ABB RobotStudio station: CellaRobot1.rspag

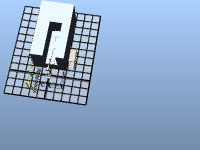
--- station ---
Station CellaRobot (saved by RobotStudio 7.0.8504.151)
Controller IRB_4600_40kg_2.55m
  mechanical unit ROB_1: IRB4600_40_255_C_01, 6 joints, base frame (0, 0, 0) mm
Layout (positions relative to the parent item):
  - IRB4600_40_255_C_01 [mechanism, from Robots\IRB4600_40_255_C_G_01.rslib] at (0, 0, 0) mm; joint values [0, 0, 0, 0, 0.5236, 0] (rad or m)
  - NHX8000 [mechanism, from ADD_Library\NHX8000.rslib] at (0, 0, 0) mm; joint values [2.6, 2] (rad or m)
  - FenceCreator [smart component, from ADD_Library\Recinzione Parametrizzabile.rslib] at (-1991.18, 2102.12, 0) mm
      properties: LengthXside1=3000; LengthYside1=-600; LengthXside2=0; LengthYside2=0; LengthYside3=0; FenceColor=Yellow
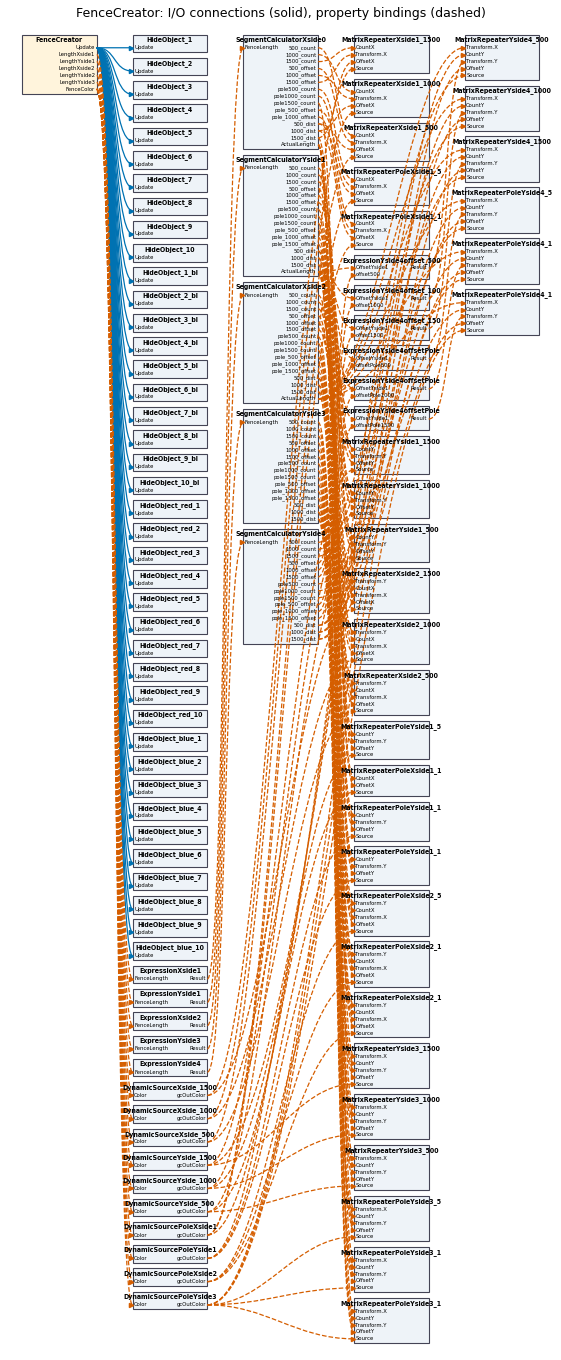
      connections:
        FenceCreator.Update -> HideObject_1.Update
        FenceCreator.Update -> HideObject_2.Update
        FenceCreator.Update -> HideObject_3.Update
        FenceCreator.Update -> HideObject_4.Update
        FenceCreator.Update -> HideObject_5.Update
        FenceCreator.Update -> HideObject_6.Update
        FenceCreator.Update -> HideObject_7.Update
        FenceCreator.Update -> HideObject_8.Update
        FenceCreator.Update -> HideObject_9.Update
        FenceCreator.Update -> HideObject_10.Update
        FenceCreator.Update -> HideObject_1_bl.Update
        FenceCreator.Update -> HideObject_2_bl.Update
        FenceCreator.Update -> HideObject_3_bl.Update
        FenceCreator.Update -> HideObject_4_bl.Update
        FenceCreator.Update -> HideObject_5_bl.Update
        FenceCreator.Update -> HideObject_6_bl.Update
        FenceCreator.Update -> HideObject_7_bl.Update
        FenceCreator.Update -> HideObject_8_bl.Update
        FenceCreator.Update -> HideObject_9_bl.Update
        FenceCreator.Update -> HideObject_10_bl.Update
        FenceCreator.Update -> HideObject_red_1.Update
        FenceCreator.Update -> HideObject_red_2.Update
        FenceCreator.Update -> HideObject_red_3.Update
        FenceCreator.Update -> HideObject_red_4.Update
        FenceCreator.Update -> HideObject_red_5.Update
        FenceCreator.Update -> HideObject_red_6.Update
        FenceCreator.Update -> HideObject_red_7.Update
        FenceCreator.Update -> HideObject_red_8.Update
        FenceCreator.Update -> HideObject_red_9.Update
        FenceCreator.Update -> HideObject_red_10.Update
        FenceCreator.Update -> HideObject_blue_1.Update
        FenceCreator.Update -> HideObject_blue_2.Update
        FenceCreator.Update -> HideObject_blue_3.Update
        FenceCreator.Update -> HideObject_blue_4.Update
        FenceCreator.Update -> HideObject_blue_5.Update
        FenceCreator.Update -> HideObject_blue_6.Update
        FenceCreator.Update -> HideObject_blue_7.Update
        FenceCreator.Update -> HideObject_blue_8.Update
        FenceCreator.Update -> HideObject_blue_9.Update
        FenceCreator.Update -> HideObject_blue_10.Update
        FenceCreator.LengthXside1 => ExpressionXside1.FenceLength
        ExpressionXside1.Result => SegmentCalculatorXside0.FenceLength
        SegmentCalculatorXside0.500_count => MatrixRepeaterXside1_500.CountX
        SegmentCalculatorXside0.1000_count => MatrixRepeaterXside1_1000.CountX
        SegmentCalculatorXside0.1500_count => MatrixRepeaterXside1_1500.CountX
        SegmentCalculatorXside0.500_offset => MatrixRepeaterXside1_500.Transform.X
        SegmentCalculatorXside0.1000_offset => MatrixRepeaterXside1_1000.Transform.X
        SegmentCalculatorXside0.1500_offset => MatrixRepeaterXside1_1500.Transform.X
        SegmentCalculatorXside0.pole500_count => MatrixRepeaterPoleXside1_500.CountX
        SegmentCalculatorXside0.pole1000_count => MatrixRepeaterPoleXside1_1000.CountX
        SegmentCalculatorXside0.pole1500_count => MatrixRepeaterPoleXside1_1500.CountX
        SegmentCalculatorXside0.pole_500_offset => MatrixRepeaterPoleXside1_500.Transform.X
        SegmentCalculatorXside0.pole_1000_offset => MatrixRepeaterPoleXside1_1000.Transform.X
        SegmentCalculatorXside0.500_dist => MatrixRepeaterXside1_500.OffsetX
        SegmentCalculatorXside0.500_dist => MatrixRepeaterPoleXside1_500.OffsetX
        SegmentCalculatorXside0.1000_dist => MatrixRepeaterXside1_1000.OffsetX
        SegmentCalculatorXside0.1000_dist => MatrixRepeaterPoleXside1_1000.OffsetX
        SegmentCalculatorXside0.1500_dist => MatrixRepeaterXside1_1500.OffsetX
        SegmentCalculatorXside0.1500_dist => MatrixRepeaterPoleXside1_1500.OffsetX
        SegmentCalculatorXside0.ActualLength => MatrixRepeaterYside3_500.Transform.X
        SegmentCalculatorXside0.ActualLength => MatrixRepeaterYside3_1000.Transform.X
        SegmentCalculatorXside0.ActualLength => MatrixRepeaterYside3_1500.Transform.X
        SegmentCalculatorXside0.ActualLength => MatrixRepeaterPoleYside3_500.Transform.X
        SegmentCalculatorXside0.ActualLength => MatrixRepeaterPoleYside3_1000.Transform.X
        SegmentCalculatorXside0.ActualLength => MatrixRepeaterPoleYside3_1500.Transform.X
        FenceCreator.LengthYside1 => ExpressionYside1.FenceLength
        ExpressionYside1.Result => SegmentCalculatorYside1.FenceLength
        SegmentCalculatorYside1.500_count => MatrixRepeaterYside1_500.CountY
        SegmentCalculatorYside1.1000_count => MatrixRepeaterYside1_1000.CountY
        SegmentCalculatorYside1.1500_count => MatrixRepeaterYside1_1500.CountY
        SegmentCalculatorYside1.500_offset => MatrixRepeaterYside1_500.Transform.Y
        SegmentCalculatorYside1.1000_offset => MatrixRepeaterYside1_1000.Transform.Y
        SegmentCalculatorYside1.1500_offset => MatrixRepeaterYside1_1500.Transform.Y
        SegmentCalculatorYside1.pole500_count => MatrixRepeaterPoleYside1_500.CountY
        SegmentCalculatorYside1.pole1000_count => MatrixRepeaterPoleYside1_1000.CountY
        SegmentCalculatorYside1.pole1500_count => MatrixRepeaterPoleYside1_1500.CountY
        SegmentCalculatorYside1.pole_500_offset => MatrixRepeaterPoleYside1_500.Transform.Y
        SegmentCalculatorYside1.pole_1000_offset => MatrixRepeaterPoleYside1_1000.Transform.Y
        SegmentCalculatorYside1.pole_1500_offset => MatrixRepeaterPoleYside1_1500.Transform.Y
        SegmentCalculatorYside1.500_dist => MatrixRepeaterYside1_500.OffsetY
        SegmentCalculatorYside1.500_dist => MatrixRepeaterPoleYside1_500.OffsetY
        SegmentCalculatorYside1.1000_dist => MatrixRepeaterYside1_1000.OffsetY
        SegmentCalculatorYside1.1000_dist => MatrixRepeaterPoleYside1_1000.OffsetY
        SegmentCalculatorYside1.1500_dist => MatrixRepeaterYside1_1500.OffsetY
        SegmentCalculatorYside1.1500_dist => MatrixRepeaterPoleYside1_1500.OffsetY
        SegmentCalculatorYside1.ActualLength => MatrixRepeaterXside2_500.Transform.Y
        SegmentCalculatorYside1.ActualLength => MatrixRepeaterXside2_1000.Transform.Y
        SegmentCalculatorYside1.ActualLength => MatrixRepeaterXside2_1500.Transform.Y
        SegmentCalculatorYside1.ActualLength => MatrixRepeaterPoleXside2_500.Transform.Y
        SegmentCalculatorYside1.ActualLength => MatrixRepeaterPoleXside2_1000.Transform.Y
        SegmentCalculatorYside1.ActualLength => MatrixRepeaterPoleXside2_1500.Transform.Y
        SegmentCalculatorYside1.ActualLength => ExpressionYside4offset_500.OffsetYside1
        SegmentCalculatorYside1.ActualLength => ExpressionYside4offset_1000.OffsetYside1
        SegmentCalculatorYside1.ActualLength => ExpressionYside4offset_1500.OffsetYside1
        SegmentCalculatorYside1.ActualLength => ExpressionYside4offsetPole_500.OffsetYside1
        SegmentCalculatorYside1.ActualLength => ExpressionYside4offsetPole_1000.OffsetYside1
        SegmentCalculatorYside1.ActualLength => ExpressionYside4offsetPole_1500.OffsetYside1
        FenceCreator.LengthXside2 => ExpressionXside2.FenceLength
        ExpressionXside2.Result => SegmentCalculatorXside2.FenceLength
        SegmentCalculatorXside2.500_count => MatrixRepeaterXside2_500.CountX
        SegmentCalculatorXside2.1000_count => MatrixRepeaterXside2_1000.CountX
        SegmentCalculatorXside2.1500_count => MatrixRepeaterXside2_1500.CountX
        SegmentCalculatorXside2.500_offset => MatrixRepeaterXside2_500.Transform.X
        SegmentCalculatorXside2.1000_offset => MatrixRepeaterXside2_1000.Transform.X
        SegmentCalculatorXside2.1500_offset => MatrixRepeaterXside2_1500.Transform.X
        SegmentCalculatorXside2.pole500_count => MatrixRepeaterPoleXside2_500.CountX
        SegmentCalculatorXside2.pole1000_count => MatrixRepeaterPoleXside2_1000.CountX
        SegmentCalculatorXside2.pole1500_count => MatrixRepeaterPoleXside2_1500.CountX
        SegmentCalculatorXside2.pole_500_offset => MatrixRepeaterPoleXside2_500.Transform.X
        SegmentCalculatorXside2.pole_1000_offset => MatrixRepeaterPoleXside2_1000.Transform.X
        SegmentCalculatorXside2.pole_1500_offset => MatrixRepeaterPoleXside2_1500.Transform.X
        SegmentCalculatorXside2.500_dist => MatrixRepeaterXside2_500.OffsetX
        SegmentCalculatorXside2.500_dist => MatrixRepeaterPoleXside2_500.OffsetX
        SegmentCalculatorXside2.1000_dist => MatrixRepeaterXside2_1000.OffsetX
        SegmentCalculatorXside2.1000_dist => MatrixRepeaterPoleXside2_1000.OffsetX
        SegmentCalculatorXside2.1500_dist => MatrixRepeaterXside2_1500.OffsetX
        SegmentCalculatorXside2.1500_dist => MatrixRepeaterPoleXside2_1500.OffsetX
        SegmentCalculatorXside2.ActualLength => MatrixRepeaterYside4_500.Transform.X
        SegmentCalculatorXside2.ActualLength => MatrixRepeaterYside4_1000.Transform.X
        SegmentCalculatorXside2.ActualLength => MatrixRepeaterYside4_1500.Transform.X
        SegmentCalculatorXside2.ActualLength => MatrixRepeaterPoleYside4_500.Transform.X
        SegmentCalculatorXside2.ActualLength => MatrixRepeaterPoleYside4_1000.Transform.X
        SegmentCalculatorXside2.ActualLength => MatrixRepeaterPoleYside4_1500.Transform.X
        FenceCreator.LengthYside2 => ExpressionYside3.FenceLength
        ExpressionYside3.Result => SegmentCalculatorYside3.FenceLength
        SegmentCalculatorYside3.500_count => MatrixRepeaterYside3_500.CountY
        SegmentCalculatorYside3.1000_count => MatrixRepeaterYside3_1000.CountY
        SegmentCalculatorYside3.1500_count => MatrixRepeaterYside3_1500.CountY
        SegmentCalculatorYside3.500_offset => MatrixRepeaterYside3_500.Transform.Y
        SegmentCalculatorYside3.1000_offset => MatrixRepeaterYside3_1000.Transform.Y
        SegmentCalculatorYside3.1500_offset => MatrixRepeaterYside3_1500.Transform.Y
        SegmentCalculatorYside3.pole500_count => MatrixRepeaterPoleYside3_500.CountY
        SegmentCalculatorYside3.pole1000_count => MatrixRepeaterPoleYside3_1000.CountY
        SegmentCalculatorYside3.pole1500_count => MatrixRepeaterPoleYside3_1500.CountY
        SegmentCalculatorYside3.pole_500_offset => MatrixRepeaterPoleYside3_500.Transform.Y
        SegmentCalculatorYside3.pole_1000_offset => MatrixRepeaterPoleYside3_1000.Transform.Y
        SegmentCalculatorYside3.pole_1500_offset => MatrixRepeaterPoleYside3_1500.Transform.Y
        SegmentCalculatorYside3.500_dist => MatrixRepeaterYside3_500.OffsetY
        SegmentCalculatorYside3.500_dist => MatrixRepeaterPoleYside3_500.OffsetY
        SegmentCalculatorYside3.1000_dist => MatrixRepeaterYside3_1000.OffsetY
        SegmentCalculatorYside3.1000_dist => MatrixRepeaterPoleYside3_1000.OffsetY
        SegmentCalculatorYside3.1500_dist => MatrixRepeaterYside3_1500.OffsetY
        SegmentCalculatorYside3.1500_dist => MatrixRepeaterPoleYside3_1500.OffsetY
        FenceCreator.LengthYside3 => ExpressionYside4.FenceLength
        ExpressionYside4.Result => SegmentCalculatorYside4.FenceLength
        SegmentCalculatorYside4.500_count => MatrixRepeaterYside4_500.CountY
        SegmentCalculatorYside4.1000_count => MatrixRepeaterYside4_1000.CountY
        SegmentCalculatorYside4.1500_count => MatrixRepeaterYside4_1500.CountY
        SegmentCalculatorYside4.500_offset => ExpressionYside4offset_500.offset500
        SegmentCalculatorYside4.1000_offset => ExpressionYside4offset_1000.offset1000
        SegmentCalculatorYside4.1500_offset => ExpressionYside4offset_1500.offset1500
        SegmentCalculatorYside4.pole500_count => MatrixRepeaterPoleYside4_500.CountY
        SegmentCalculatorYside4.pole1000_count => MatrixRepeaterPoleYside4_1000.CountY
        SegmentCalculatorYside4.pole1500_count => MatrixRepeaterPoleYside4_1500.CountY
        SegmentCalculatorYside4.pole_500_offset => ExpressionYside4offsetPole_500.offsetPole500
        SegmentCalculatorYside4.pole_1000_offset => ExpressionYside4offsetPole_1000.offsetPole1000
        SegmentCalculatorYside4.pole_1500_offset => ExpressionYside4offsetPole_1500.offsetPole1500
        ExpressionYside4offset_500.Result => MatrixRepeaterYside4_500.Transform.Y
        ExpressionYside4offset_1000.Result => MatrixRepeaterYside4_1000.Transform.Y
        ExpressionYside4offset_1500.Result => MatrixRepeaterYside4_1500.Transform.Y
        ExpressionYside4offsetPole_500.Result => MatrixRepeaterPoleYside4_500.Transform.Y
        ExpressionYside4offsetPole_1000.Result => MatrixRepeaterPoleYside4_1000.Transform.Y
        ExpressionYside4offsetPole_1500.Result => MatrixRepeaterPoleYside4_1500.Transform.Y
        SegmentCalculatorYside4.500_dist => MatrixRepeaterYside4_500.OffsetY
        SegmentCalculatorYside4.500_dist => MatrixRepeaterPoleYside4_500.OffsetY
        SegmentCalculatorYside4.1000_dist => MatrixRepeaterYside4_1000.OffsetY
        SegmentCalculatorYside4.1000_dist => MatrixRepeaterPoleYside4_1000.OffsetY
        SegmentCalculatorYside4.1500_dist => MatrixRepeaterYside4_1500.OffsetY
        SegmentCalculatorYside4.1500_dist => MatrixRepeaterPoleYside4_1500.OffsetY
        FenceCreator.FenceColor => DynamicSourceXside_1500.Color
        DynamicSourceXside_1500.gcOutColor => MatrixRepeaterXside1_1500.Source
        DynamicSourceXside_1500.gcOutColor => MatrixRepeaterXside2_1500.Source
        FenceCreator.FenceColor => DynamicSourceXside_1000.Color
        DynamicSourceXside_1000.gcOutColor => MatrixRepeaterXside1_1000.Source
        DynamicSourceXside_1000.gcOutColor => MatrixRepeaterXside2_1000.Source
        FenceCreator.FenceColor => DynamicSourceXside_500.Color
        DynamicSourceXside_500.gcOutColor => MatrixRepeaterXside1_500.Source
        DynamicSourceXside_500.gcOutColor => MatrixRepeaterXside2_500.Source
        FenceCreator.FenceColor => DynamicSourceYside_1500.Color
        DynamicSourceYside_1500.gcOutColor => MatrixRepeaterYside1_1500.Source
        DynamicSourceYside_1500.gcOutColor => MatrixRepeaterYside3_1500.Source
        DynamicSourceYside_1500.gcOutColor => MatrixRepeaterYside4_1500.Source
        FenceCreator.FenceColor => DynamicSourceYside_1000.Color
        DynamicSourceYside_1000.gcOutColor => MatrixRepeaterYside1_1000.Source
        DynamicSourceYside_1000.gcOutColor => MatrixRepeaterYside3_1000.Source
        DynamicSourceYside_1000.gcOutColor => MatrixRepeaterYside4_1000.Source
        FenceCreator.FenceColor => DynamicSourceYside_500.Color
        DynamicSourceYside_500.gcOutColor => MatrixRepeaterYside1_500.Source
        DynamicSourceYside_500.gcOutColor => MatrixRepeaterYside3_500.Source
        DynamicSourceYside_500.gcOutColor => MatrixRepeaterYside4_500.Source
        FenceCreator.FenceColor => DynamicSourcePoleXside1.Color
        DynamicSourcePoleXside1.gcOutColor => MatrixRepeaterPoleXside1_1500.Source
        DynamicSourcePoleXside1.gcOutColor => MatrixRepeaterPoleXside1_1000.Source
        DynamicSourcePoleXside1.gcOutColor => MatrixRepeaterPoleXside1_500.Source
        FenceCreator.FenceColor => DynamicSourcePoleYside1.Color
        DynamicSourcePoleYside1.gcOutColor => MatrixRepeaterPoleYside1_1500.Source
        DynamicSourcePoleYside1.gcOutColor => MatrixRepeaterPoleYside1_1000.Source
        DynamicSourcePoleYside1.gcOutColor => MatrixRepeaterPoleYside1_500.Source
        FenceCreator.FenceColor => DynamicSourcePoleXside2.Color
        DynamicSourcePoleXside2.gcOutColor => MatrixRepeaterPoleXside2_1500.Source
        DynamicSourcePoleXside2.gcOutColor => MatrixRepeaterPoleXside2_1000.Source
        DynamicSourcePoleXside2.gcOutColor => MatrixRepeaterPoleXside2_500.Source
        FenceCreator.FenceColor => DynamicSourcePoleYside3.Color
        DynamicSourcePoleYside3.gcOutColor => MatrixRepeaterPoleYside3_1500.Source
        DynamicSourcePoleYside3.gcOutColor => MatrixRepeaterPoleYside3_1000.Source
        DynamicSourcePoleYside3.gcOutColor => MatrixRepeaterPoleYside3_500.Source
        DynamicSourcePoleYside3.gcOutColor => MatrixRepeaterPoleYside4_1500.Source
        DynamicSourcePoleYside3.gcOutColor => MatrixRepeaterPoleYside4_1000.Source
        DynamicSourcePoleYside3.gcOutColor => MatrixRepeaterPoleYside4_500.Source
    - ExpressionXside1 [smart component, from ADD_Library\Recinzione Parametrizzabile.rslib]
        properties: Expression=FenceLength/1000; Result=3; FenceLength=3000
    - MatrixRepeaterXside1_1500 [smart component, from ADD_Library\Recinzione Parametrizzabile.rslib]
        properties: Source=Panel 2000x1500 X ye; CountX=2; CountY=1; CountZ=1; OffsetX=1.5; OffsetY=0; OffsetZ=0
      - Panel 2000x1500 X ye [part, from ADD_Library\Recinzione Parametrizzabile.rslib]
      - Panel 2000x1500 X ye [part, from ADD_Library\Recinzione Parametrizzabile.rslib] at (1500, 0, 0) mm
    - Panel 2000x1000 X ye [part, from ADD_Library\Recinzione Parametrizzabile.rslib]
    - Panel 2000x500 X ye [part, from ADD_Library\Recinzione Parametrizzabile.rslib]
    - Panel 2000x1500 X ye [part, from ADD_Library\Recinzione Parametrizzabile.rslib]
    - MatrixRepeaterXside1_1000 [smart component, from ADD_Library\Recinzione Parametrizzabile.rslib] at (3000, 0, 0) mm
        properties: Source=Panel 2000x1000 X ye; CountX=0; CountY=1; CountZ=1; OffsetX=1; OffsetY=0; OffsetZ=0
    - MatrixRepeaterXside1_500 [smart component, from ADD_Library\Recinzione Parametrizzabile.rslib] at (3000, 0, 0) mm
        properties: Source=Panel 2000x500 X ye; CountX=0; CountY=1; CountZ=1; OffsetX=0.5; OffsetY=0; OffsetZ=0
    - MatrixRepeaterPoleXside1_1000 [smart component, from ADD_Library\Recinzione Parametrizzabile.rslib] at (4000, 0, 0) mm
        properties: Source=Pole ye; CountX=0; CountY=1; CountZ=1; OffsetX=1; OffsetY=0; OffsetZ=0
    - Pole ye [part, from ADD_Library\Recinzione Parametrizzabile.rslib]
    - SegmentCalculatorXside0 [smart component, from ADD_Library\Recinzione Parametrizzabile.rslib]
        properties: FenceLength=3; ActualLength=3; 1500_dist=1.5; 1000_dist=1; 500_dist=0.5; 1500_offset=0; 1000_offset=3; 500_offset=3; pole_1500_offset=0; pole_1000_offset=4; pole_500_offset=3.5; 1500_count=2; 1000_count=0; 500_count=0; pole1500_count=3; pole1000_count=0; pole500_count=0; SideNo=0
    - MatrixRepeaterPoleXside1_1500 [smart component, from ADD_Library\Recinzione Parametrizzabile.rslib]
        properties: Source=Pole ye; CountX=3; CountY=1; CountZ=1; OffsetX=1.5; OffsetY=0; OffsetZ=1
      - Pole ye [part, from ADD_Library\Recinzione Parametrizzabile.rslib]
      - Pole ye [part, from ADD_Library\Recinzione Parametrizzabile.rslib] at (1500, 0, 0) mm
      - Pole ye [part, from ADD_Library\Recinzione Parametrizzabile.rslib] at (3000, 0, 0) mm
    - MatrixRepeaterPoleXside1_500 [smart component, from ADD_Library\Recinzione Parametrizzabile.rslib] at (3500, 0, 0) mm
        properties: Source=Pole ye; CountX=0; CountY=1; CountZ=1; OffsetX=0.5; OffsetY=0; OffsetZ=0
    - Panel 2000x1000 Y ye [part, from ADD_Library\Recinzione Parametrizzabile.rslib]
    - Panel 2000x500 Y ye [part, from ADD_Library\Recinzione Parametrizzabile.rslib]
    - Panel 2000x1500 Y ye [part, from ADD_Library\Recinzione Parametrizzabile.rslib]
    - ExpressionYside1 [smart component, from ADD_Library\Recinzione Parametrizzabile.rslib]
        properties: Expression=FenceLength/1000; Result=-0.6; FenceLength=-600
    - MatrixRepeaterYside1_1500 [smart component, from ADD_Library\Recinzione Parametrizzabile.rslib] at (0, -1500, 0) mm
        properties: Source=Panel 2000x1500 Y ye; CountX=1; CountY=0; CountZ=1; OffsetX=0; OffsetY=-1.5; OffsetZ=0
    - MatrixRepeaterYside1_1000 [smart component, from ADD_Library\Recinzione Parametrizzabile.rslib] at (0, -1000, 0) mm
        properties: Source=Panel 2000x1000 Y ye; CountX=1; CountY=0; CountZ=1; OffsetX=0; OffsetY=-1; OffsetZ=0
    - MatrixRepeaterYside1_500 [smart component, from ADD_Library\Recinzione Parametrizzabile.rslib] at (0, -500, 0) mm
        properties: Source=Panel 2000x500 Y ye; CountX=1; CountY=1; CountZ=1; OffsetX=0; OffsetY=-0.5; OffsetZ=0
      - Panel 2000x500 Y ye [part, from ADD_Library\Recinzione Parametrizzabile.rslib]
    - PoleYside1 ye [part, from ADD_Library\Recinzione Parametrizzabile.rslib]
    - MatrixRepeaterPoleYside1_1500 [smart component, from ADD_Library\Recinzione Parametrizzabile.rslib] at (0, 1500, 0) mm
        properties: Source=PoleYside1 ye; CountX=1; CountY=0; CountZ=1; OffsetX=0; OffsetY=-1.5; OffsetZ=0
    - SegmentCalculatorYside1 [smart component, from ADD_Library\Recinzione Parametrizzabile.rslib]
        properties: FenceLength=-0.6; ActualLength=-0.5; 1500_dist=-1.5; 1000_dist=-1; 500_dist=-0.5; 1500_offset=-1.5; 1000_offset=-1; 500_offset=-0.5; pole_1500_offset=1.5; pole_1000_offset=1; pole_500_offset=-0.5; 1500_count=0; 1000_count=0; 500_count=1; pole1500_count=0; pole1000_count=0; pole500_count=1; SideNo=1
    - MatrixRepeaterPoleYside1_1000 [smart component, from ADD_Library\Recinzione Parametrizzabile.rslib] at (0, 1000, 0) mm
        properties: Source=PoleYside1 ye; CountX=1; CountY=0; CountZ=1; OffsetX=0; OffsetY=-1; OffsetZ=0
    - MatrixRepeaterPoleYside1_500 [smart component, from ADD_Library\Recinzione Parametrizzabile.rslib] at (0, -500, 0) mm
        properties: Source=PoleYside1 ye; CountX=1; CountY=1; CountZ=1; OffsetX=0; OffsetY=-0.5; OffsetZ=0
      - PoleYside1 ye [part, from ADD_Library\Recinzione Parametrizzabile.rslib]
    - PoleXside2 ye [part, from ADD_Library\Recinzione Parametrizzabile.rslib]
    - PoleYside3 ye [part, from ADD_Library\Recinzione Parametrizzabile.rslib]
    - ExpressionXside2 [smart component, from ADD_Library\Recinzione Parametrizzabile.rslib]
        properties: Expression=FenceLength/1000; Result=0; FenceLength=0
    - SegmentCalculatorXside2 [smart component, from ADD_Library\Recinzione Parametrizzabile.rslib]
        properties: FenceLength=0; ActualLength=0; 1500_dist=1.5; 1000_dist=1; 500_dist=0.5; 1500_offset=0; 1000_offset=0; 500_offset=0; pole_1500_offset=1.5; pole_1000_offset=1; pole_500_offset=0; 1500_count=0; 1000_count=0; 500_count=0; pole1500_count=0; pole1000_count=0; pole500_count=0; SideNo=2
    - MatrixRepeaterXside2_1500 [smart component, from ADD_Library\Recinzione Parametrizzabile.rslib] at (0, -500, 0) mm
        properties: Source=Panel 2000x1500 X ye; CountX=0; CountY=1; CountZ=1; OffsetX=1.5; OffsetY=0; OffsetZ=0
    - MatrixRepeaterXside2_1000 [smart component, from ADD_Library\Recinzione Parametrizzabile.rslib] at (0, -500, 0) mm
        properties: Source=Panel 2000x1000 X ye; CountX=0; CountY=1; CountZ=1; OffsetX=1; OffsetY=0; OffsetZ=0
    - MatrixRepeaterXside2_500 [smart component, from ADD_Library\Recinzione Parametrizzabile.rslib] at (0, -500, 0) mm
        properties: Source=Panel 2000x500 X ye; CountX=0; CountY=1; CountZ=1; OffsetX=0.5; OffsetY=0; OffsetZ=0
    - MatrixRepeaterPoleXside2_1500 [smart component, from ADD_Library\Recinzione Parametrizzabile.rslib] at (1500, -500, 0) mm
        properties: Source=PoleXside2 ye; CountX=0; CountY=1; CountZ=1; OffsetX=1.5; OffsetY=0; OffsetZ=0
    - MatrixRepeaterPoleXside2_1000 [smart component, from ADD_Library\Recinzione Parametrizzabile.rslib] at (1000, -500, 0) mm
        properties: Source=PoleXside2 ye; CountX=0; CountY=1; CountZ=1; OffsetX=1; OffsetY=0; OffsetZ=0
    - MatrixRepeaterPoleXside2_500 [smart component, from ADD_Library\Recinzione Parametrizzabile.rslib] at (0, -500, 0) mm
        properties: Source=PoleXside2 ye; CountX=0; CountY=1; CountZ=1; OffsetX=0.5; OffsetY=0; OffsetZ=0
    - SegmentCalculatorYside3 [smart component, from ADD_Library\Recinzione Parametrizzabile.rslib]
        properties: FenceLength=0; ActualLength=0; 1500_dist=1.5; 1000_dist=1; 500_dist=0.5; 1500_offset=0; 1000_offset=0; 500_offset=0; pole_1500_offset=-1.5; pole_1000_offset=-2.5; pole_500_offset=0; 1500_count=0; 1000_count=0; 500_count=0; pole1500_count=0; pole1000_count=0; pole500_count=0; SideNo=3
    - ExpressionYside3 [smart component, from ADD_Library\Recinzione Parametrizzabile.rslib]
        properties: Expression=FenceLength/1000; Result=0; FenceLength=0
    - MatrixRepeaterYside3_1500 [smart component, from ADD_Library\Recinzione Parametrizzabile.rslib] at (3000, 0, 0) mm
        properties: Source=Panel 2000x1500 Y ye; CountX=1; CountY=0; CountZ=1; OffsetX=0; OffsetY=1.5; OffsetZ=0
    - MatrixRepeaterYside3_1000 [smart component, from ADD_Library\Recinzione Parametrizzabile.rslib] at (3000, 0, 0) mm
        properties: Source=Panel 2000x1000 Y ye; CountX=1; CountY=0; CountZ=1; OffsetX=0; OffsetY=1; OffsetZ=0
    - MatrixRepeaterYside3_500 [smart component, from ADD_Library\Recinzione Parametrizzabile.rslib] at (3000, 0, 0) mm
        properties: Source=Panel 2000x500 Y ye; CountX=1; CountY=0; CountZ=1; OffsetX=0; OffsetY=0.5; OffsetZ=0
    - MatrixRepeaterPoleYside3_1500 [smart component, from ADD_Library\Recinzione Parametrizzabile.rslib] at (3000, -1500, 0) mm
        properties: Source=PoleYside3 ye; CountX=1; CountY=0; CountZ=1; OffsetX=0; OffsetY=1.5; OffsetZ=0
    - MatrixRepeaterPoleYside3_1000 [smart component, from ADD_Library\Recinzione Parametrizzabile.rslib] at (3000, -2500, 0) mm
        properties: Source=PoleYside3 ye; CountX=1; CountY=0; CountZ=1; OffsetX=0; OffsetY=1; OffsetZ=0
    - MatrixRepeaterPoleYside3_500 [smart component, from ADD_Library\Recinzione Parametrizzabile.rslib] at (3000, 0, 0) mm
        properties: Source=PoleYside3 ye; CountX=1; CountY=0; CountZ=1; OffsetX=0; OffsetY=0.5; OffsetZ=0
    - ExpressionYside4 [smart component, from ADD_Library\Recinzione Parametrizzabile.rslib]
        properties: Expression=FenceLength/1000; Result=0; FenceLength=0
    - SegmentCalculatorYside4 [smart component, from ADD_Library\Recinzione Parametrizzabile.rslib]
        properties: FenceLength=0; ActualLength=0; 1500_dist=1.5; 1000_dist=1; 500_dist=0.5; 1500_offset=0; 1000_offset=0; 500_offset=0; pole_1500_offset=1.5; pole_1000_offset=2.5; pole_500_offset=0; 1500_count=0; 1000_count=0; 500_count=0; pole1500_count=0; pole1000_count=0; pole500_count=0; SideNo=4
    - MatrixRepeaterYside4_1500 [smart component, from ADD_Library\Recinzione Parametrizzabile.rslib] at (0, -500, 0) mm
        properties: Source=Panel 2000x1500 Y ye; CountX=1; CountY=0; CountZ=1; OffsetX=0; OffsetY=1.5; OffsetZ=0
    - ExpressionYside4offset_500 [smart component, from ADD_Library\Recinzione Parametrizzabile.rslib]
        properties: Expression=OffsetYside1+offset500; Result=-0.5; OffsetYside1=-0.5; offset500=0
    - ExpressionYside4offset_1000 [smart component, from ADD_Library\Recinzione Parametrizzabile.rslib]
        properties: Expression=OffsetYside1+offset1000; Result=-0.5; OffsetYside1=-0.5; offset1000=0
    - ExpressionYside4offset_1500 [smart component, from ADD_Library\Recinzione Parametrizzabile.rslib]
        properties: Expression=OffsetYside1+offset1500; Result=-0.5; OffsetYside1=-0.5; offset1500=0
    - MatrixRepeaterYside4_1000 [smart component, from ADD_Library\Recinzione Parametrizzabile.rslib] at (0, -500, 0) mm
        properties: Source=Panel 2000x1000 Y ye; CountX=1; CountY=0; CountZ=1; OffsetX=0; OffsetY=1; OffsetZ=0
    - MatrixRepeaterYside4_500 [smart component, from ADD_Library\Recinzione Parametrizzabile.rslib] at (0, -500, 0) mm
        properties: Source=Panel 2000x500 Y ye; CountX=1; CountY=0; CountZ=1; OffsetX=0; OffsetY=0.5; OffsetZ=0
    - ExpressionYside4offsetPole_500 [smart component, from ADD_Library\Recinzione Parametrizzabile.rslib]
        properties: Expression=OffsetYside1+offsetPole500; Result=-0.5; OffsetYside1=-0.5; offsetPole500=0
    - ExpressionYside4offsetPole_1000 [smart component, from ADD_Library\Recinzione Parametrizzabile.rslib]
        properties: Expression=OffsetYside1+offsetPole1000; Result=2; OffsetYside1=-0.5; offsetPole1000=2.5
    - ExpressionYside4offsetPole_1500 [smart component, from ADD_Library\Recinzione Parametrizzabile.rslib]
        properties: Expression=OffsetYside1+offsetPole1500; Result=1; OffsetYside1=-0.5; offsetPole1500=1.5
    - MatrixRepeaterPoleYside4_500 [smart component, from ADD_Library\Recinzione Parametrizzabile.rslib] at (0, -500, 0) mm
        properties: Source=PoleYside3 ye; CountX=1; CountY=0; CountZ=1; OffsetX=0; OffsetY=0.5; OffsetZ=0
    - MatrixRepeaterPoleYside4_1000 [smart component, from ADD_Library\Recinzione Parametrizzabile.rslib] at (0, 2000, 0) mm
        properties: Source=PoleYside3 ye; CountX=1; CountY=0; CountZ=1; OffsetX=0; OffsetY=1; OffsetZ=0
    - MatrixRepeaterPoleYside4_1500 [smart component, from ADD_Library\Recinzione Parametrizzabile.rslib] at (0, 1000, 0) mm
        properties: Source=PoleYside3 ye; CountX=1; CountY=0; CountZ=1; OffsetX=0; OffsetY=1.5; OffsetZ=0
    - HideObject_1 [smart component, from ADD_Library\Recinzione Parametrizzabile.rslib]
        properties: Object=Panel 2000x500 X ye
    - HideObject_2 [smart component, from ADD_Library\Recinzione Parametrizzabile.rslib]
        properties: Object=Panel 2000x1000 X ye
    - HideObject_3 [smart component, from ADD_Library\Recinzione Parametrizzabile.rslib]
        properties: Object=Panel 2000x1500 X ye
    - HideObject_4 [smart component, from ADD_Library\Recinzione Parametrizzabile.rslib]
        properties: Object=Panel 2000x500 Y ye
    - HideObject_5 [smart component, from ADD_Library\Recinzione Parametrizzabile.rslib]
        properties: Object=Panel 2000x1000 Y ye
    - HideObject_6 [smart component, from ADD_Library\Recinzione Parametrizzabile.rslib]
        properties: Object=Panel 2000x1500 Y ye
    - HideObject_7 [smart component, from ADD_Library\Recinzione Parametrizzabile.rslib]
        properties: Object=Pole ye
    - HideObject_8 [smart component, from ADD_Library\Recinzione Parametrizzabile.rslib]
        properties: Object=PoleYside1 ye
    - HideObject_9 [smart component, from ADD_Library\Recinzione Parametrizzabile.rslib]
        properties: Object=PoleXside2 ye
    - HideObject_10 [smart component, from ADD_Library\Recinzione Parametrizzabile.rslib]
        properties: Object=PoleYside3 ye
    - Panel 2000x1000 X bl [part, from ADD_Library\Recinzione Parametrizzabile.rslib]
    - Panel 2000x500 X bl [part, from ADD_Library\Recinzione Parametrizzabile.rslib]
    - Panel 2000x1500 X bl [part, from ADD_Library\Recinzione Parametrizzabile.rslib]
    - Pole bl [part, from ADD_Library\Recinzione Parametrizzabile.rslib]
    - Panel 2000x1000 Y bl [part, from ADD_Library\Recinzione Parametrizzabile.rslib]
    - Panel 2000x500 Y bl [part, from ADD_Library\Recinzione Parametrizzabile.rslib]
    - Panel 2000x1500 Y bl [part, from ADD_Library\Recinzione Parametrizzabile.rslib]
    - PoleYside1 bl [part, from ADD_Library\Recinzione Parametrizzabile.rslib]
    - PoleXside2 bl [part, from ADD_Library\Recinzione Parametrizzabile.rslib]
    - PoleYside3 bl [part, from ADD_Library\Recinzione Parametrizzabile.rslib]
    - DynamicSourceXside_1500 [smart component, from ADD_Library\Recinzione Parametrizzabile.rslib]
        properties: gcBlack=Panel 2000x1500 X bl; gcYellow=Panel 2000x1500 X ye; gcRed=Panel 2000x1500 X red; gcBlue=Panel 2000x1500 X_blue; Color=Yellow; gcOutColor=Panel 2000x1500 X ye
    - DynamicSourceXside_1000 [smart component, from ADD_Library\Recinzione Parametrizzabile.rslib]
        properties: gcBlack=Panel 2000x1000 X bl; gcYellow=Panel 2000x1000 X ye; gcRed=Panel 2000x1000 X red; gcBlue=Panel 2000x1000 X_blue; Color=Yellow; gcOutColor=Panel 2000x1000 X ye
    - DynamicSourceXside_500 [smart component, from ADD_Library\Recinzione Parametrizzabile.rslib]
        properties: gcBlack=Panel 2000x500 X bl; gcYellow=Panel 2000x500 X ye; gcRed=Panel 2000x500 X red; gcBlue=Panel 2000x500 X blue; Color=Yellow; gcOutColor=Panel 2000x500 X ye
    - DynamicSourceYside_1500 [smart component, from ADD_Library\Recinzione Parametrizzabile.rslib]
        properties: gcBlack=Panel 2000x1500 Y bl; gcYellow=Panel 2000x1500 Y ye; gcRed=Panel 2000x1500 Y red; gcBlue=Panel 2000x1500 Y_blue; Color=Yellow; gcOutColor=Panel 2000x1500 Y ye
    - DynamicSourceYside_1000 [smart component, from ADD_Library\Recinzione Parametrizzabile.rslib]
        properties: gcBlack=Panel 2000x1000 Y bl; gcYellow=Panel 2000x1000 Y ye; gcRed=Panel 2000x1000 Y red; gcBlue=Panel 2000x1000 Y_blue; Color=Yellow; gcOutColor=Panel 2000x1000 Y ye
    - DynamicSourceYside_500 [smart component, from ADD_Library\Recinzione Parametrizzabile.rslib]
        properties: gcBlack=Panel 2000x500 Y bl; gcYellow=Panel 2000x500 Y ye; gcRed=Panel 2000x500 Y red; gcBlue=Panel 2000x500 Y blue; Color=Yellow; gcOutColor=Panel 2000x500 Y ye
    - DynamicSourcePoleXside1 [smart component, from ADD_Library\Recinzione Parametrizzabile.rslib]
        properties: gcBlack=Pole bl; gcYellow=Pole ye; gcRed=Pole_red; gcBlue=Pole_blue; Color=Yellow; gcOutColor=Pole ye
    - DynamicSourcePoleYside1 [smart component, from ADD_Library\Recinzione Parametrizzabile.rslib]
        properties: gcBlack=PoleYside1 bl; gcYellow=PoleYside1 ye; gcRed=PoleYside1_red; gcBlue=PoleYside1_blue; Color=Yellow; gcOutColor=PoleYside1 ye
    - DynamicSourcePoleXside2 [smart component, from ADD_Library\Recinzione Parametrizzabile.rslib]
        properties: gcBlack=PoleXside2 bl; gcYellow=PoleXside2 ye; gcRed=PoleXside2_red; gcBlue=PoleXside2_blue; Color=Yellow; gcOutColor=PoleXside2 ye
    - DynamicSourcePoleYside3 [smart component, from ADD_Library\Recinzione Parametrizzabile.rslib]
        properties: gcBlack=PoleYside3 bl; gcYellow=PoleYside3 ye; gcRed=PoleYside3 red; gcBlue=PoleYside3 blue; Color=Yellow; gcOutColor=PoleYside3 ye
    - HideObject_1_bl [smart component, from ADD_Library\Recinzione Parametrizzabile.rslib]
        properties: Object=Panel 2000x1500 X bl
    - HideObject_2_bl [smart component, from ADD_Library\Recinzione Parametrizzabile.rslib]
        properties: Object=Panel 2000x1000 X bl
    - HideObject_3_bl [smart component, from ADD_Library\Recinzione Parametrizzabile.rslib]
        properties: Object=Panel 2000x500 X bl
    - HideObject_4_bl [smart component, from ADD_Library\Recinzione Parametrizzabile.rslib]
        properties: Object=Panel 2000x1500 Y bl
    - HideObject_5_bl [smart component, from ADD_Library\Recinzione Parametrizzabile.rslib]
        properties: Object=Panel 2000x1000 Y bl
    - HideObject_6_bl [smart component, from ADD_Library\Recinzione Parametrizzabile.rslib]
        properties: Object=Panel 2000x500 Y bl
    - HideObject_7_bl [smart component, from ADD_Library\Recinzione Parametrizzabile.rslib]
        properties: Object=Pole bl
    - HideObject_8_bl [smart component, from ADD_Library\Recinzione Parametrizzabile.rslib]
        properties: Object=PoleYside1 bl
    - HideObject_9_bl [smart component, from ADD_Library\Recinzione Parametrizzabile.rslib]
        properties: Object=PoleXside2 bl
    - HideObject_10_bl [smart component, from ADD_Library\Recinzione Parametrizzabile.rslib]
        properties: Object=PoleYside3 bl
    - Panel 2000x500 X blue [part, from ADD_Library\Recinzione Parametrizzabile.rslib]
    - Panel 2000x500 X red [part, from ADD_Library\Recinzione Parametrizzabile.rslib]
    - Panel 2000x500 Y blue [part, from ADD_Library\Recinzione Parametrizzabile.rslib]
    - Panel 2000x500 Y red [part, from ADD_Library\Recinzione Parametrizzabile.rslib]
    - Panel 2000x1000 X red [part, from ADD_Library\Recinzione Parametrizzabile.rslib]
    - Panel 2000x1000 X_blue [part, from ADD_Library\Recinzione Parametrizzabile.rslib]
    - Panel 2000x1000 Y red [part, from ADD_Library\Recinzione Parametrizzabile.rslib]
    - Panel 2000x1000 Y_blue [part, from ADD_Library\Recinzione Parametrizzabile.rslib]
    - Panel 2000x1500 X red [part, from ADD_Library\Recinzione Parametrizzabile.rslib]
    - Panel 2000x1500 X_blue [part, from ADD_Library\Recinzione Parametrizzabile.rslib]
    - Panel 2000x1500 Y red [part, from ADD_Library\Recinzione Parametrizzabile.rslib]
    - Panel 2000x1500 Y_blue [part, from ADD_Library\Recinzione Parametrizzabile.rslib]
    - Pole_blue [part, from ADD_Library\Recinzione Parametrizzabile.rslib]
    - Pole_red [part, from ADD_Library\Recinzione Parametrizzabile.rslib]
    - PoleXside2_blue [part, from ADD_Library\Recinzione Parametrizzabile.rslib]
    - PoleXside2_red [part, from ADD_Library\Recinzione Parametrizzabile.rslib]
    - PoleYside1_blue [part, from ADD_Library\Recinzione Parametrizzabile.rslib]
    - PoleYside1_red [part, from ADD_Library\Recinzione Parametrizzabile.rslib]
    - PoleYside3 blue [part, from ADD_Library\Recinzione Parametrizzabile.rslib]
    - PoleYside3 red [part, from ADD_Library\Recinzione Parametrizzabile.rslib]
    - HideObject_red_1 [smart component, from ADD_Library\Recinzione Parametrizzabile.rslib]
        properties: Object=Panel 2000x1500 X red
    - HideObject_red_2 [smart component, from ADD_Library\Recinzione Parametrizzabile.rslib]
        properties: Object=Panel 2000x1500 Y red
    - HideObject_red_3 [smart component, from ADD_Library\Recinzione Parametrizzabile.rslib]
        properties: Object=Panel 2000x1000 X red
    - HideObject_red_4 [smart component, from ADD_Library\Recinzione Parametrizzabile.rslib]
        properties: Object=Panel 2000x1000 Y red
    - HideObject_red_5 [smart component, from ADD_Library\Recinzione Parametrizzabile.rslib]
        properties: Object=Panel 2000x500 X red
    - HideObject_red_6 [smart component, from ADD_Library\Recinzione Parametrizzabile.rslib]
        properties: Object=Panel 2000x500 Y red
    - HideObject_red_7 [smart component, from ADD_Library\Recinzione Parametrizzabile.rslib]
        properties: Object=Pole_red
    - HideObject_red_8 [smart component, from ADD_Library\Recinzione Parametrizzabile.rslib]
        properties: Object=PoleXside2_red
    - HideObject_red_9 [smart component, from ADD_Library\Recinzione Parametrizzabile.rslib]
        properties: Object=PoleYside1_red
    - HideObject_red_10 [smart component, from ADD_Library\Recinzione Parametrizzabile.rslib]
        properties: Object=PoleYside3 red
    - HideObject_blue_1 [smart component, from ADD_Library\Recinzione Parametrizzabile.rslib]
        properties: Object=Panel 2000x1500 X_blue
    - HideObject_blue_2 [smart component, from ADD_Library\Recinzione Parametrizzabile.rslib]
        properties: Object=Panel 2000x1500 Y_blue
    - HideObject_blue_3 [smart component, from ADD_Library\Recinzione Parametrizzabile.rslib]
        properties: Object=Panel 2000x1000 X_blue
    - HideObject_blue_4 [smart component, from ADD_Library\Recinzione Parametrizzabile.rslib]
        properties: Object=Panel 2000x1000 Y_blue
    - HideObject_blue_5 [smart component, from ADD_Library\Recinzione Parametrizzabile.rslib]
        properties: Object=Panel 2000x500 X blue
    - HideObject_blue_6 [smart component, from ADD_Library\Recinzione Parametrizzabile.rslib]
        properties: Object=Panel 2000x500 Y blue
    - HideObject_blue_7 [smart component, from ADD_Library\Recinzione Parametrizzabile.rslib]
        properties: Object=Pole_blue
    - HideObject_blue_8 [smart component, from ADD_Library\Recinzione Parametrizzabile.rslib]
        properties: Object=PoleXside2_blue
    - HideObject_blue_9 [smart component, from ADD_Library\Recinzione Parametrizzabile.rslib]
        properties: Object=PoleYside1_blue
    - HideObject_blue_10 [smart component, from ADD_Library\Recinzione Parametrizzabile.rslib]
        properties: Object=PoleYside3 blue
  - FenceCreator_2 [smart component, from ADD_Library\Recinzione Parametrizzabile.rslib] at (-1501.5, -1896.94, 0) mm
      properties: LengthXside1=2500; LengthYside1=2500; LengthXside2=0; LengthYside2=0; LengthYside3=0; FenceColor=Black
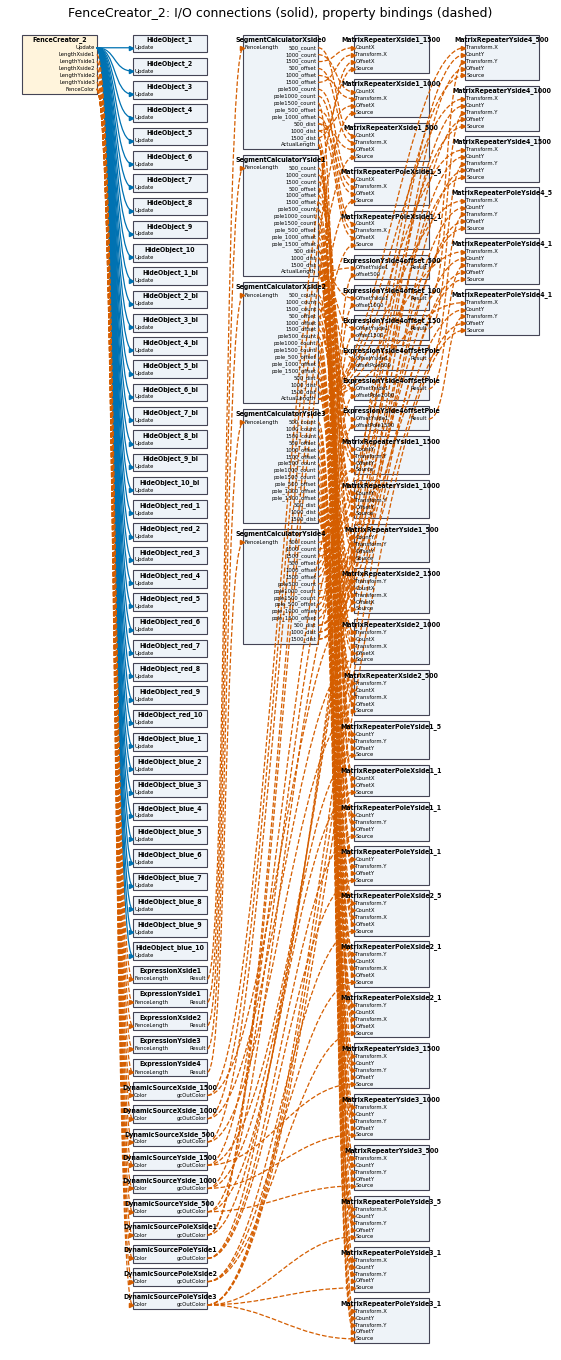
      connections:
        FenceCreator_2.Update -> HideObject_1.Update
        FenceCreator_2.Update -> HideObject_2.Update
        FenceCreator_2.Update -> HideObject_3.Update
        FenceCreator_2.Update -> HideObject_4.Update
        FenceCreator_2.Update -> HideObject_5.Update
        FenceCreator_2.Update -> HideObject_6.Update
        FenceCreator_2.Update -> HideObject_7.Update
        FenceCreator_2.Update -> HideObject_8.Update
        FenceCreator_2.Update -> HideObject_9.Update
        FenceCreator_2.Update -> HideObject_10.Update
        FenceCreator_2.Update -> HideObject_1_bl.Update
        FenceCreator_2.Update -> HideObject_2_bl.Update
        FenceCreator_2.Update -> HideObject_3_bl.Update
        FenceCreator_2.Update -> HideObject_4_bl.Update
        FenceCreator_2.Update -> HideObject_5_bl.Update
        FenceCreator_2.Update -> HideObject_6_bl.Update
        FenceCreator_2.Update -> HideObject_7_bl.Update
        FenceCreator_2.Update -> HideObject_8_bl.Update
        FenceCreator_2.Update -> HideObject_9_bl.Update
        FenceCreator_2.Update -> HideObject_10_bl.Update
        FenceCreator_2.Update -> HideObject_red_1.Update
        FenceCreator_2.Update -> HideObject_red_2.Update
        FenceCreator_2.Update -> HideObject_red_3.Update
        FenceCreator_2.Update -> HideObject_red_4.Update
        FenceCreator_2.Update -> HideObject_red_5.Update
        FenceCreator_2.Update -> HideObject_red_6.Update
        FenceCreator_2.Update -> HideObject_red_7.Update
        FenceCreator_2.Update -> HideObject_red_8.Update
        FenceCreator_2.Update -> HideObject_red_9.Update
        FenceCreator_2.Update -> HideObject_red_10.Update
        FenceCreator_2.Update -> HideObject_blue_1.Update
        FenceCreator_2.Update -> HideObject_blue_2.Update
        FenceCreator_2.Update -> HideObject_blue_3.Update
        FenceCreator_2.Update -> HideObject_blue_4.Update
        FenceCreator_2.Update -> HideObject_blue_5.Update
        FenceCreator_2.Update -> HideObject_blue_6.Update
        FenceCreator_2.Update -> HideObject_blue_7.Update
        FenceCreator_2.Update -> HideObject_blue_8.Update
        FenceCreator_2.Update -> HideObject_blue_9.Update
        FenceCreator_2.Update -> HideObject_blue_10.Update
        FenceCreator_2.LengthXside1 => ExpressionXside1.FenceLength
        ExpressionXside1.Result => SegmentCalculatorXside0.FenceLength
        SegmentCalculatorXside0.500_count => MatrixRepeaterXside1_500.CountX
        SegmentCalculatorXside0.1000_count => MatrixRepeaterXside1_1000.CountX
        SegmentCalculatorXside0.1500_count => MatrixRepeaterXside1_1500.CountX
        SegmentCalculatorXside0.500_offset => MatrixRepeaterXside1_500.Transform.X
        SegmentCalculatorXside0.1000_offset => MatrixRepeaterXside1_1000.Transform.X
        SegmentCalculatorXside0.1500_offset => MatrixRepeaterXside1_1500.Transform.X
        SegmentCalculatorXside0.pole500_count => MatrixRepeaterPoleXside1_500.CountX
        SegmentCalculatorXside0.pole1000_count => MatrixRepeaterPoleXside1_1000.CountX
        SegmentCalculatorXside0.pole1500_count => MatrixRepeaterPoleXside1_1500.CountX
        SegmentCalculatorXside0.pole_500_offset => MatrixRepeaterPoleXside1_500.Transform.X
        SegmentCalculatorXside0.pole_1000_offset => MatrixRepeaterPoleXside1_1000.Transform.X
        SegmentCalculatorXside0.500_dist => MatrixRepeaterXside1_500.OffsetX
        SegmentCalculatorXside0.500_dist => MatrixRepeaterPoleXside1_500.OffsetX
        SegmentCalculatorXside0.1000_dist => MatrixRepeaterXside1_1000.OffsetX
        SegmentCalculatorXside0.1000_dist => MatrixRepeaterPoleXside1_1000.OffsetX
        SegmentCalculatorXside0.1500_dist => MatrixRepeaterXside1_1500.OffsetX
        SegmentCalculatorXside0.1500_dist => MatrixRepeaterPoleXside1_1500.OffsetX
        SegmentCalculatorXside0.ActualLength => MatrixRepeaterYside3_500.Transform.X
        SegmentCalculatorXside0.ActualLength => MatrixRepeaterYside3_1000.Transform.X
        SegmentCalculatorXside0.ActualLength => MatrixRepeaterYside3_1500.Transform.X
        SegmentCalculatorXside0.ActualLength => MatrixRepeaterPoleYside3_500.Transform.X
        SegmentCalculatorXside0.ActualLength => MatrixRepeaterPoleYside3_1000.Transform.X
        SegmentCalculatorXside0.ActualLength => MatrixRepeaterPoleYside3_1500.Transform.X
        FenceCreator_2.LengthYside1 => ExpressionYside1.FenceLength
        ExpressionYside1.Result => SegmentCalculatorYside1.FenceLength
        SegmentCalculatorYside1.500_count => MatrixRepeaterYside1_500.CountY
        SegmentCalculatorYside1.1000_count => MatrixRepeaterYside1_1000.CountY
        SegmentCalculatorYside1.1500_count => MatrixRepeaterYside1_1500.CountY
        SegmentCalculatorYside1.500_offset => MatrixRepeaterYside1_500.Transform.Y
        SegmentCalculatorYside1.1000_offset => MatrixRepeaterYside1_1000.Transform.Y
        SegmentCalculatorYside1.1500_offset => MatrixRepeaterYside1_1500.Transform.Y
        SegmentCalculatorYside1.pole500_count => MatrixRepeaterPoleYside1_500.CountY
        SegmentCalculatorYside1.pole1000_count => MatrixRepeaterPoleYside1_1000.CountY
        SegmentCalculatorYside1.pole1500_count => MatrixRepeaterPoleYside1_1500.CountY
        SegmentCalculatorYside1.pole_500_offset => MatrixRepeaterPoleYside1_500.Transform.Y
        SegmentCalculatorYside1.pole_1000_offset => MatrixRepeaterPoleYside1_1000.Transform.Y
        SegmentCalculatorYside1.pole_1500_offset => MatrixRepeaterPoleYside1_1500.Transform.Y
        SegmentCalculatorYside1.500_dist => MatrixRepeaterYside1_500.OffsetY
        SegmentCalculatorYside1.500_dist => MatrixRepeaterPoleYside1_500.OffsetY
        SegmentCalculatorYside1.1000_dist => MatrixRepeaterYside1_1000.OffsetY
        SegmentCalculatorYside1.1000_dist => MatrixRepeaterPoleYside1_1000.OffsetY
        SegmentCalculatorYside1.1500_dist => MatrixRepeaterYside1_1500.OffsetY
        SegmentCalculatorYside1.1500_dist => MatrixRepeaterPoleYside1_1500.OffsetY
        SegmentCalculatorYside1.ActualLength => MatrixRepeaterXside2_500.Transform.Y
        SegmentCalculatorYside1.ActualLength => MatrixRepeaterXside2_1000.Transform.Y
        SegmentCalculatorYside1.ActualLength => MatrixRepeaterXside2_1500.Transform.Y
        SegmentCalculatorYside1.ActualLength => MatrixRepeaterPoleXside2_500.Transform.Y
        SegmentCalculatorYside1.ActualLength => MatrixRepeaterPoleXside2_1000.Transform.Y
        SegmentCalculatorYside1.ActualLength => MatrixRepeaterPoleXside2_1500.Transform.Y
        SegmentCalculatorYside1.ActualLength => ExpressionYside4offset_500.OffsetYside1
        SegmentCalculatorYside1.ActualLength => ExpressionYside4offset_1000.OffsetYside1
        SegmentCalculatorYside1.ActualLength => ExpressionYside4offset_1500.OffsetYside1
        SegmentCalculatorYside1.ActualLength => ExpressionYside4offsetPole_500.OffsetYside1
        SegmentCalculatorYside1.ActualLength => ExpressionYside4offsetPole_1000.OffsetYside1
        SegmentCalculatorYside1.ActualLength => ExpressionYside4offsetPole_1500.OffsetYside1
        FenceCreator_2.LengthXside2 => ExpressionXside2.FenceLength
        ExpressionXside2.Result => SegmentCalculatorXside2.FenceLength
        SegmentCalculatorXside2.500_count => MatrixRepeaterXside2_500.CountX
        SegmentCalculatorXside2.1000_count => MatrixRepeaterXside2_1000.CountX
        SegmentCalculatorXside2.1500_count => MatrixRepeaterXside2_1500.CountX
        SegmentCalculatorXside2.500_offset => MatrixRepeaterXside2_500.Transform.X
        SegmentCalculatorXside2.1000_offset => MatrixRepeaterXside2_1000.Transform.X
        SegmentCalculatorXside2.1500_offset => MatrixRepeaterXside2_1500.Transform.X
        SegmentCalculatorXside2.pole500_count => MatrixRepeaterPoleXside2_500.CountX
        SegmentCalculatorXside2.pole1000_count => MatrixRepeaterPoleXside2_1000.CountX
        SegmentCalculatorXside2.pole1500_count => MatrixRepeaterPoleXside2_1500.CountX
        SegmentCalculatorXside2.pole_500_offset => MatrixRepeaterPoleXside2_500.Transform.X
        SegmentCalculatorXside2.pole_1000_offset => MatrixRepeaterPoleXside2_1000.Transform.X
        SegmentCalculatorXside2.pole_1500_offset => MatrixRepeaterPoleXside2_1500.Transform.X
        SegmentCalculatorXside2.500_dist => MatrixRepeaterXside2_500.OffsetX
        SegmentCalculatorXside2.500_dist => MatrixRepeaterPoleXside2_500.OffsetX
        SegmentCalculatorXside2.1000_dist => MatrixRepeaterXside2_1000.OffsetX
        SegmentCalculatorXside2.1000_dist => MatrixRepeaterPoleXside2_1000.OffsetX
        SegmentCalculatorXside2.1500_dist => MatrixRepeaterXside2_1500.OffsetX
        SegmentCalculatorXside2.1500_dist => MatrixRepeaterPoleXside2_1500.OffsetX
        SegmentCalculatorXside2.ActualLength => MatrixRepeaterYside4_500.Transform.X
        SegmentCalculatorXside2.ActualLength => MatrixRepeaterYside4_1000.Transform.X
        SegmentCalculatorXside2.ActualLength => MatrixRepeaterYside4_1500.Transform.X
        SegmentCalculatorXside2.ActualLength => MatrixRepeaterPoleYside4_500.Transform.X
        SegmentCalculatorXside2.ActualLength => MatrixRepeaterPoleYside4_1000.Transform.X
        SegmentCalculatorXside2.ActualLength => MatrixRepeaterPoleYside4_1500.Transform.X
        FenceCreator_2.LengthYside2 => ExpressionYside3.FenceLength
        ExpressionYside3.Result => SegmentCalculatorYside3.FenceLength
        SegmentCalculatorYside3.500_count => MatrixRepeaterYside3_500.CountY
        SegmentCalculatorYside3.1000_count => MatrixRepeaterYside3_1000.CountY
        SegmentCalculatorYside3.1500_count => MatrixRepeaterYside3_1500.CountY
        SegmentCalculatorYside3.500_offset => MatrixRepeaterYside3_500.Transform.Y
        SegmentCalculatorYside3.1000_offset => MatrixRepeaterYside3_1000.Transform.Y
        SegmentCalculatorYside3.1500_offset => MatrixRepeaterYside3_1500.Transform.Y
        SegmentCalculatorYside3.pole500_count => MatrixRepeaterPoleYside3_500.CountY
        SegmentCalculatorYside3.pole1000_count => MatrixRepeaterPoleYside3_1000.CountY
        SegmentCalculatorYside3.pole1500_count => MatrixRepeaterPoleYside3_1500.CountY
        SegmentCalculatorYside3.pole_500_offset => MatrixRepeaterPoleYside3_500.Transform.Y
        SegmentCalculatorYside3.pole_1000_offset => MatrixRepeaterPoleYside3_1000.Transform.Y
        SegmentCalculatorYside3.pole_1500_offset => MatrixRepeaterPoleYside3_1500.Transform.Y
        SegmentCalculatorYside3.500_dist => MatrixRepeaterYside3_500.OffsetY
        SegmentCalculatorYside3.500_dist => MatrixRepeaterPoleYside3_500.OffsetY
        SegmentCalculatorYside3.1000_dist => MatrixRepeaterYside3_1000.OffsetY
        SegmentCalculatorYside3.1000_dist => MatrixRepeaterPoleYside3_1000.OffsetY
        SegmentCalculatorYside3.1500_dist => MatrixRepeaterYside3_1500.OffsetY
        SegmentCalculatorYside3.1500_dist => MatrixRepeaterPoleYside3_1500.OffsetY
        FenceCreator_2.LengthYside3 => ExpressionYside4.FenceLength
        ExpressionYside4.Result => SegmentCalculatorYside4.FenceLength
        SegmentCalculatorYside4.500_count => MatrixRepeaterYside4_500.CountY
        SegmentCalculatorYside4.1000_count => MatrixRepeaterYside4_1000.CountY
        SegmentCalculatorYside4.1500_count => MatrixRepeaterYside4_1500.CountY
        SegmentCalculatorYside4.500_offset => ExpressionYside4offset_500.offset500
        SegmentCalculatorYside4.1000_offset => ExpressionYside4offset_1000.offset1000
        SegmentCalculatorYside4.1500_offset => ExpressionYside4offset_1500.offset1500
        SegmentCalculatorYside4.pole500_count => MatrixRepeaterPoleYside4_500.CountY
        SegmentCalculatorYside4.pole1000_count => MatrixRepeaterPoleYside4_1000.CountY
        SegmentCalculatorYside4.pole1500_count => MatrixRepeaterPoleYside4_1500.CountY
        SegmentCalculatorYside4.pole_500_offset => ExpressionYside4offsetPole_500.offsetPole500
        SegmentCalculatorYside4.pole_1000_offset => ExpressionYside4offsetPole_1000.offsetPole1000
        SegmentCalculatorYside4.pole_1500_offset => ExpressionYside4offsetPole_1500.offsetPole1500
        ExpressionYside4offset_500.Result => MatrixRepeaterYside4_500.Transform.Y
        ExpressionYside4offset_1000.Result => MatrixRepeaterYside4_1000.Transform.Y
        ExpressionYside4offset_1500.Result => MatrixRepeaterYside4_1500.Transform.Y
        ExpressionYside4offsetPole_500.Result => MatrixRepeaterPoleYside4_500.Transform.Y
        ExpressionYside4offsetPole_1000.Result => MatrixRepeaterPoleYside4_1000.Transform.Y
        ExpressionYside4offsetPole_1500.Result => MatrixRepeaterPoleYside4_1500.Transform.Y
        SegmentCalculatorYside4.500_dist => MatrixRepeaterYside4_500.OffsetY
        SegmentCalculatorYside4.500_dist => MatrixRepeaterPoleYside4_500.OffsetY
        SegmentCalculatorYside4.1000_dist => MatrixRepeaterYside4_1000.OffsetY
        SegmentCalculatorYside4.1000_dist => MatrixRepeaterPoleYside4_1000.OffsetY
        SegmentCalculatorYside4.1500_dist => MatrixRepeaterYside4_1500.OffsetY
        SegmentCalculatorYside4.1500_dist => MatrixRepeaterPoleYside4_1500.OffsetY
        FenceCreator_2.FenceColor => DynamicSourceXside_1500.Color
        DynamicSourceXside_1500.gcOutColor => MatrixRepeaterXside1_1500.Source
        DynamicSourceXside_1500.gcOutColor => MatrixRepeaterXside2_1500.Source
        FenceCreator_2.FenceColor => DynamicSourceXside_1000.Color
        DynamicSourceXside_1000.gcOutColor => MatrixRepeaterXside1_1000.Source
        DynamicSourceXside_1000.gcOutColor => MatrixRepeaterXside2_1000.Source
        FenceCreator_2.FenceColor => DynamicSourceXside_500.Color
        DynamicSourceXside_500.gcOutColor => MatrixRepeaterXside1_500.Source
        DynamicSourceXside_500.gcOutColor => MatrixRepeaterXside2_500.Source
        FenceCreator_2.FenceColor => DynamicSourceYside_1500.Color
        DynamicSourceYside_1500.gcOutColor => MatrixRepeaterYside1_1500.Source
        DynamicSourceYside_1500.gcOutColor => MatrixRepeaterYside3_1500.Source
        DynamicSourceYside_1500.gcOutColor => MatrixRepeaterYside4_1500.Source
        FenceCreator_2.FenceColor => DynamicSourceYside_1000.Color
        DynamicSourceYside_1000.gcOutColor => MatrixRepeaterYside1_1000.Source
        DynamicSourceYside_1000.gcOutColor => MatrixRepeaterYside3_1000.Source
        DynamicSourceYside_1000.gcOutColor => MatrixRepeaterYside4_1000.Source
        FenceCreator_2.FenceColor => DynamicSourceYside_500.Color
        DynamicSourceYside_500.gcOutColor => MatrixRepeaterYside1_500.Source
        DynamicSourceYside_500.gcOutColor => MatrixRepeaterYside3_500.Source
        DynamicSourceYside_500.gcOutColor => MatrixRepeaterYside4_500.Source
        FenceCreator_2.FenceColor => DynamicSourcePoleXside1.Color
        DynamicSourcePoleXside1.gcOutColor => MatrixRepeaterPoleXside1_1500.Source
        DynamicSourcePoleXside1.gcOutColor => MatrixRepeaterPoleXside1_1000.Source
        DynamicSourcePoleXside1.gcOutColor => MatrixRepeaterPoleXside1_500.Source
        FenceCreator_2.FenceColor => DynamicSourcePoleYside1.Color
        DynamicSourcePoleYside1.gcOutColor => MatrixRepeaterPoleYside1_1500.Source
        DynamicSourcePoleYside1.gcOutColor => MatrixRepeaterPoleYside1_1000.Source
        DynamicSourcePoleYside1.gcOutColor => MatrixRepeaterPoleYside1_500.Source
        FenceCreator_2.FenceColor => DynamicSourcePoleXside2.Color
        DynamicSourcePoleXside2.gcOutColor => MatrixRepeaterPoleXside2_1500.Source
        DynamicSourcePoleXside2.gcOutColor => MatrixRepeaterPoleXside2_1000.Source
        DynamicSourcePoleXside2.gcOutColor => MatrixRepeaterPoleXside2_500.Source
        FenceCreator_2.FenceColor => DynamicSourcePoleYside3.Color
        DynamicSourcePoleYside3.gcOutColor => MatrixRepeaterPoleYside3_1500.Source
        DynamicSourcePoleYside3.gcOutColor => MatrixRepeaterPoleYside3_1000.Source
        DynamicSourcePoleYside3.gcOutColor => MatrixRepeaterPoleYside3_500.Source
        DynamicSourcePoleYside3.gcOutColor => MatrixRepeaterPoleYside4_1500.Source
        DynamicSourcePoleYside3.gcOutColor => MatrixRepeaterPoleYside4_1000.Source
        DynamicSourcePoleYside3.gcOutColor => MatrixRepeaterPoleYside4_500.Source
    - ExpressionXside1 [smart component, from ADD_Library\Recinzione Parametrizzabile.rslib]
        properties: Expression=FenceLength/1000; Result=2.5; FenceLength=2500
    - MatrixRepeaterXside1_1500 [smart component, from ADD_Library\Recinzione Parametrizzabile.rslib]
        properties: Source=Panel 2000x1500 X bl; CountX=1; CountY=1; CountZ=1; OffsetX=1.5; OffsetY=0; OffsetZ=0
      - Panel 2000x1500 X bl [part, from ADD_Library\Recinzione Parametrizzabile.rslib]
    - Panel 2000x1000 X ye [part, from ADD_Library\Recinzione Parametrizzabile.rslib]
    - Panel 2000x500 X ye [part, from ADD_Library\Recinzione Parametrizzabile.rslib]
    - Panel 2000x1500 X ye [part, from ADD_Library\Recinzione Parametrizzabile.rslib]
    - MatrixRepeaterXside1_1000 [smart component, from ADD_Library\Recinzione Parametrizzabile.rslib] at (1500, 0, 0) mm
        properties: Source=Panel 2000x1000 X bl; CountX=1; CountY=1; CountZ=1; OffsetX=1; OffsetY=0; OffsetZ=0
      - Panel 2000x1000 X bl [part, from ADD_Library\Recinzione Parametrizzabile.rslib]
    - MatrixRepeaterXside1_500 [smart component, from ADD_Library\Recinzione Parametrizzabile.rslib] at (2500, 0, 0) mm
        properties: Source=Panel 2000x500 X bl; CountX=0; CountY=1; CountZ=1; OffsetX=0.5; OffsetY=0; OffsetZ=0
    - MatrixRepeaterPoleXside1_1000 [smart component, from ADD_Library\Recinzione Parametrizzabile.rslib] at (2500, 0, 0) mm
        properties: Source=Pole bl; CountX=1; CountY=1; CountZ=1; OffsetX=1; OffsetY=0; OffsetZ=0
      - Pole bl [part, from ADD_Library\Recinzione Parametrizzabile.rslib]
    - Pole ye [part, from ADD_Library\Recinzione Parametrizzabile.rslib]
    - SegmentCalculatorXside0 [smart component, from ADD_Library\Recinzione Parametrizzabile.rslib]
        properties: FenceLength=2.5; ActualLength=2.5; 1500_dist=1.5; 1000_dist=1; 500_dist=0.5; 1500_offset=0; 1000_offset=1.5; 500_offset=2.5; pole_1500_offset=0; pole_1000_offset=2.5; pole_500_offset=3; 1500_count=1; 1000_count=1; 500_count=0; pole1500_count=2; pole1000_count=1; pole500_count=0; SideNo=0
    - MatrixRepeaterPoleXside1_1500 [smart component, from ADD_Library\Recinzione Parametrizzabile.rslib]
        properties: Source=Pole bl; CountX=2; CountY=1; CountZ=1; OffsetX=1.5; OffsetY=0; OffsetZ=1
      - Pole bl [part, from ADD_Library\Recinzione Parametrizzabile.rslib]
      - Pole bl [part, from ADD_Library\Recinzione Parametrizzabile.rslib] at (1500, 0, 0) mm
    - MatrixRepeaterPoleXside1_500 [smart component, from ADD_Library\Recinzione Parametrizzabile.rslib] at (3000, 0, 0) mm
        properties: Source=Pole bl; CountX=0; CountY=1; CountZ=1; OffsetX=0.5; OffsetY=0; OffsetZ=0
    - Panel 2000x1000 Y ye [part, from ADD_Library\Recinzione Parametrizzabile.rslib]
    - Panel 2000x500 Y ye [part, from ADD_Library\Recinzione Parametrizzabile.rslib]
    - Panel 2000x1500 Y ye [part, from ADD_Library\Recinzione Parametrizzabile.rslib]
    - ExpressionYside1 [smart component, from ADD_Library\Recinzione Parametrizzabile.rslib]
        properties: Expression=FenceLength/1000; Result=2.5; FenceLength=2500
    - MatrixRepeaterYside1_1500 [smart component, from ADD_Library\Recinzione Parametrizzabile.rslib]
        properties: Source=Panel 2000x1500 Y bl; CountX=1; CountY=1; CountZ=1; OffsetX=0; OffsetY=1.5; OffsetZ=0
      - Panel 2000x1500 Y bl [part, from ADD_Library\Recinzione Parametrizzabile.rslib]
    - MatrixRepeaterYside1_1000 [smart component, from ADD_Library\Recinzione Parametrizzabile.rslib] at (0, 1500, 0) mm
        properties: Source=Panel 2000x1000 Y bl; CountX=1; CountY=1; CountZ=1; OffsetX=0; OffsetY=1; OffsetZ=0
      - Panel 2000x1000 Y bl [part, from ADD_Library\Recinzione Parametrizzabile.rslib]
    - MatrixRepeaterYside1_500 [smart component, from ADD_Library\Recinzione Parametrizzabile.rslib] at (0, 2500, 0) mm
        properties: Source=Panel 2000x500 Y bl; CountX=1; CountY=0; CountZ=1; OffsetX=0; OffsetY=0.5; OffsetZ=0
    - PoleYside1 ye [part, from ADD_Library\Recinzione Parametrizzabile.rslib]
    - MatrixRepeaterPoleYside1_1500 [smart component, from ADD_Library\Recinzione Parametrizzabile.rslib] at (0, 1500, 0) mm
        properties: Source=PoleYside1 bl; CountX=1; CountY=1; CountZ=1; OffsetX=0; OffsetY=1.5; OffsetZ=0
      - PoleYside1 bl [part, from ADD_Library\Recinzione Parametrizzabile.rslib]
    - SegmentCalculatorYside1 [smart component, from ADD_Library\Recinzione Parametrizzabile.rslib]
        properties: FenceLength=2.5; ActualLength=2.5; 1500_dist=1.5; 1000_dist=1; 500_dist=0.5; 1500_offset=0; 1000_offset=1.5; 500_offset=2.5; pole_1500_offset=1.5; pole_1000_offset=2.5; pole_500_offset=3; 1500_count=1; 1000_count=1; 500_count=0; pole1500_count=1; pole1000_count=1; pole500_count=0; SideNo=1
    - MatrixRepeaterPoleYside1_1000 [smart component, from ADD_Library\Recinzione Parametrizzabile.rslib] at (0, 2500, 0) mm
        properties: Source=PoleYside1 bl; CountX=1; CountY=1; CountZ=1; OffsetX=0; OffsetY=1; OffsetZ=0
      - PoleYside1 bl [part, from ADD_Library\Recinzione Parametrizzabile.rslib]
    - MatrixRepeaterPoleYside1_500 [smart component, from ADD_Library\Recinzione Parametrizzabile.rslib] at (0, 3000, 0) mm
        properties: Source=PoleYside1 bl; CountX=1; CountY=0; CountZ=1; OffsetX=0; OffsetY=0.5; OffsetZ=0
    - PoleXside2 ye [part, from ADD_Library\Recinzione Parametrizzabile.rslib]
    - PoleYside3 ye [part, from ADD_Library\Recinzione Parametrizzabile.rslib]
    - ExpressionXside2 [smart component, from ADD_Library\Recinzione Parametrizzabile.rslib]
        properties: Expression=FenceLength/1000; Result=0; FenceLength=0
    - SegmentCalculatorXside2 [smart component, from ADD_Library\Recinzione Parametrizzabile.rslib]
        properties: FenceLength=0; ActualLength=0; 1500_dist=1.5; 1000_dist=1; 500_dist=0.5; 1500_offset=0; 1000_offset=0; 500_offset=0; pole_1500_offset=1.5; pole_1000_offset=1; pole_500_offset=0; 1500_count=0; 1000_count=0; 500_count=0; pole1500_count=0; pole1000_count=0; pole500_count=0; SideNo=2
    - MatrixRepeaterXside2_1500 [smart component, from ADD_Library\Recinzione Parametrizzabile.rslib] at (0, 2500, 0) mm
        properties: Source=Panel 2000x1500 X bl; CountX=0; CountY=1; CountZ=1; OffsetX=1.5; OffsetY=0; OffsetZ=0
    - MatrixRepeaterXside2_1000 [smart component, from ADD_Library\Recinzione Parametrizzabile.rslib] at (0, 2500, 0) mm
        properties: Source=Panel 2000x1000 X bl; CountX=0; CountY=1; CountZ=1; OffsetX=1; OffsetY=0; OffsetZ=0
    - MatrixRepeaterXside2_500 [smart component, from ADD_Library\Recinzione Parametrizzabile.rslib] at (0, 2500, 0) mm
        properties: Source=Panel 2000x500 X bl; CountX=0; CountY=1; CountZ=1; OffsetX=0.5; OffsetY=0; OffsetZ=0
    - MatrixRepeaterPoleXside2_1500 [smart component, from ADD_Library\Recinzione Parametrizzabile.rslib] at (1500, 2500, 0) mm
        properties: Source=PoleXside2 bl; CountX=0; CountY=1; CountZ=1; OffsetX=1.5; OffsetY=0; OffsetZ=0
    - MatrixRepeaterPoleXside2_1000 [smart component, from ADD_Library\Recinzione Parametrizzabile.rslib] at (1000, 2500, 0) mm
        properties: Source=PoleXside2 bl; CountX=0; CountY=1; CountZ=1; OffsetX=1; OffsetY=0; OffsetZ=0
    - MatrixRepeaterPoleXside2_500 [smart component, from ADD_Library\Recinzione Parametrizzabile.rslib] at (0, 2500, 0) mm
        properties: Source=PoleXside2 bl; CountX=0; CountY=1; CountZ=1; OffsetX=0.5; OffsetY=0; OffsetZ=0
    - SegmentCalculatorYside3 [smart component, from ADD_Library\Recinzione Parametrizzabile.rslib]
        properties: FenceLength=0; ActualLength=0; 1500_dist=1.5; 1000_dist=1; 500_dist=0.5; 1500_offset=0; 1000_offset=0; 500_offset=0; pole_1500_offset=-1.5; pole_1000_offset=-2.5; pole_500_offset=0; 1500_count=0; 1000_count=0; 500_count=0; pole1500_count=0; pole1000_count=0; pole500_count=0; SideNo=3
    - ExpressionYside3 [smart component, from ADD_Library\Recinzione Parametrizzabile.rslib]
        properties: Expression=FenceLength/1000; Result=0; FenceLength=0
    - MatrixRepeaterYside3_1500 [smart component, from ADD_Library\Recinzione Parametrizzabile.rslib] at (2500, 0, 0) mm
        properties: Source=Panel 2000x1500 Y bl; CountX=1; CountY=0; CountZ=1; OffsetX=0; OffsetY=1.5; OffsetZ=0
    - MatrixRepeaterYside3_1000 [smart component, from ADD_Library\Recinzione Parametrizzabile.rslib] at (2500, 0, 0) mm
        properties: Source=Panel 2000x1000 Y bl; CountX=1; CountY=0; CountZ=1; OffsetX=0; OffsetY=1; OffsetZ=0
    - MatrixRepeaterYside3_500 [smart component, from ADD_Library\Recinzione Parametrizzabile.rslib] at (2500, 0, 0) mm
        properties: Source=Panel 2000x500 Y bl; CountX=1; CountY=0; CountZ=1; OffsetX=0; OffsetY=0.5; OffsetZ=0
    - MatrixRepeaterPoleYside3_1500 [smart component, from ADD_Library\Recinzione Parametrizzabile.rslib] at (2500, -1500, 0) mm
        properties: Source=PoleYside3 bl; CountX=1; CountY=0; CountZ=1; OffsetX=0; OffsetY=1.5; OffsetZ=0
    - MatrixRepeaterPoleYside3_1000 [smart component, from ADD_Library\Recinzione Parametrizzabile.rslib] at (2500, -2500, 0) mm
        properties: Source=PoleYside3 bl; CountX=1; CountY=0; CountZ=1; OffsetX=0; OffsetY=1; OffsetZ=0
    - MatrixRepeaterPoleYside3_500 [smart component, from ADD_Library\Recinzione Parametrizzabile.rslib] at (2500, 0, 0) mm
        properties: Source=PoleYside3 bl; CountX=1; CountY=0; CountZ=1; OffsetX=0; OffsetY=0.5; OffsetZ=0
    - ExpressionYside4 [smart component, from ADD_Library\Recinzione Parametrizzabile.rslib]
        properties: Expression=FenceLength/1000; Result=0; FenceLength=0
    - SegmentCalculatorYside4 [smart component, from ADD_Library\Recinzione Parametrizzabile.rslib]
        properties: FenceLength=0; ActualLength=0; 1500_dist=1.5; 1000_dist=1; 500_dist=0.5; 1500_offset=0; 1000_offset=0; 500_offset=0; pole_1500_offset=1.5; pole_1000_offset=2.5; pole_500_offset=0; 1500_count=0; 1000_count=0; 500_count=0; pole1500_count=0; pole1000_count=0; pole500_count=0; SideNo=4
    - MatrixRepeaterYside4_1500 [smart component, from ADD_Library\Recinzione Parametrizzabile.rslib] at (0, 2500, 0) mm
        properties: Source=Panel 2000x1500 Y bl; CountX=1; CountY=0; CountZ=1; OffsetX=0; OffsetY=1.5; OffsetZ=0
    - ExpressionYside4offset_500 [smart component, from ADD_Library\Recinzione Parametrizzabile.rslib]
        properties: Expression=OffsetYside1+offset500; Result=2.5; OffsetYside1=2.5; offset500=0
    - ExpressionYside4offset_1000 [smart component, from ADD_Library\Recinzione Parametrizzabile.rslib]
        properties: Expression=OffsetYside1+offset1000; Result=2.5; OffsetYside1=2.5; offset1000=0
    - ExpressionYside4offset_1500 [smart component, from ADD_Library\Recinzione Parametrizzabile.rslib]
        properties: Expression=OffsetYside1+offset1500; Result=2.5; OffsetYside1=2.5; offset1500=0
    - MatrixRepeaterYside4_1000 [smart component, from ADD_Library\Recinzione Parametrizzabile.rslib] at (0, 2500, 0) mm
        properties: Source=Panel 2000x1000 Y bl; CountX=1; CountY=0; CountZ=1; OffsetX=0; OffsetY=1; OffsetZ=0
    - MatrixRepeaterYside4_500 [smart component, from ADD_Library\Recinzione Parametrizzabile.rslib] at (0, 2500, 0) mm
        properties: Source=Panel 2000x500 Y bl; CountX=1; CountY=0; CountZ=1; OffsetX=0; OffsetY=0.5; OffsetZ=0
    - ExpressionYside4offsetPole_500 [smart component, from ADD_Library\Recinzione Parametrizzabile.rslib]
        properties: Expression=OffsetYside1+offsetPole500; Result=2.5; OffsetYside1=2.5; offsetPole500=0
    - ExpressionYside4offsetPole_1000 [smart component, from ADD_Library\Recinzione Parametrizzabile.rslib]
        properties: Expression=OffsetYside1+offsetPole1000; Result=5; OffsetYside1=2.5; offsetPole1000=2.5
    - ExpressionYside4offsetPole_1500 [smart component, from ADD_Library\Recinzione Parametrizzabile.rslib]
        properties: Expression=OffsetYside1+offsetPole1500; Result=4; OffsetYside1=2.5; offsetPole1500=1.5
    - MatrixRepeaterPoleYside4_500 [smart component, from ADD_Library\Recinzione Parametrizzabile.rslib] at (0, 2500, 0) mm
        properties: Source=PoleYside3 bl; CountX=1; CountY=0; CountZ=1; OffsetX=0; OffsetY=0.5; OffsetZ=0
    - MatrixRepeaterPoleYside4_1000 [smart component, from ADD_Library\Recinzione Parametrizzabile.rslib] at (0, 5000, 0) mm
        properties: Source=PoleYside3 bl; CountX=1; CountY=0; CountZ=1; OffsetX=0; OffsetY=1; OffsetZ=0
    - MatrixRepeaterPoleYside4_1500 [smart component, from ADD_Library\Recinzione Parametrizzabile.rslib] at (0, 4000, 0) mm
        properties: Source=PoleYside3 bl; CountX=1; CountY=0; CountZ=1; OffsetX=0; OffsetY=1.5; OffsetZ=0
    - HideObject_1 [smart component, from ADD_Library\Recinzione Parametrizzabile.rslib]
        properties: Object=Panel 2000x500 X ye
    - HideObject_2 [smart component, from ADD_Library\Recinzione Parametrizzabile.rslib]
        properties: Object=Panel 2000x1000 X ye
    - HideObject_3 [smart component, from ADD_Library\Recinzione Parametrizzabile.rslib]
        properties: Object=Panel 2000x1500 X ye
    - HideObject_4 [smart component, from ADD_Library\Recinzione Parametrizzabile.rslib]
        properties: Object=Panel 2000x500 Y ye
    - HideObject_5 [smart component, from ADD_Library\Recinzione Parametrizzabile.rslib]
        properties: Object=Panel 2000x1000 Y ye
    - HideObject_6 [smart component, from ADD_Library\Recinzione Parametrizzabile.rslib]
        properties: Object=Panel 2000x1500 Y ye
    - HideObject_7 [smart component, from ADD_Library\Recinzione Parametrizzabile.rslib]
        properties: Object=Pole ye
    - HideObject_8 [smart component, from ADD_Library\Recinzione Parametrizzabile.rslib]
        properties: Object=PoleYside1 ye
    - HideObject_9 [smart component, from ADD_Library\Recinzione Parametrizzabile.rslib]
        properties: Object=PoleXside2 ye
    - HideObject_10 [smart component, from ADD_Library\Recinzione Parametrizzabile.rslib]
        properties: Object=PoleYside3 ye
    - Panel 2000x1000 X bl [part, from ADD_Library\Recinzione Parametrizzabile.rslib]
    - Panel 2000x500 X bl [part, from ADD_Library\Recinzione Parametrizzabile.rslib]
    - Panel 2000x1500 X bl [part, from ADD_Library\Recinzione Parametrizzabile.rslib]
    - Pole bl [part, from ADD_Library\Recinzione Parametrizzabile.rslib]
    - Panel 2000x1000 Y bl [part, from ADD_Library\Recinzione Parametrizzabile.rslib]
    - Panel 2000x500 Y bl [part, from ADD_Library\Recinzione Parametrizzabile.rslib]
    - Panel 2000x1500 Y bl [part, from ADD_Library\Recinzione Parametrizzabile.rslib]
    - PoleYside1 bl [part, from ADD_Library\Recinzione Parametrizzabile.rslib]
    - PoleXside2 bl [part, from ADD_Library\Recinzione Parametrizzabile.rslib]
    - PoleYside3 bl [part, from ADD_Library\Recinzione Parametrizzabile.rslib]
    - DynamicSourceXside_1500 [smart component, from ADD_Library\Recinzione Parametrizzabile.rslib]
        properties: gcBlack=Panel 2000x1500 X bl; gcYellow=Panel 2000x1500 X ye; gcRed=Panel 2000x1500 X red; gcBlue=Panel 2000x1500 X_blue; Color=Black; gcOutColor=Panel 2000x1500 X bl
    - DynamicSourceXside_1000 [smart component, from ADD_Library\Recinzione Parametrizzabile.rslib]
        properties: gcBlack=Panel 2000x1000 X bl; gcYellow=Panel 2000x1000 X ye; gcRed=Panel 2000x1000 X red; gcBlue=Panel 2000x1000 X_blue; Color=Black; gcOutColor=Panel 2000x1000 X bl
    - DynamicSourceXside_500 [smart component, from ADD_Library\Recinzione Parametrizzabile.rslib]
        properties: gcBlack=Panel 2000x500 X bl; gcYellow=Panel 2000x500 X ye; gcRed=Panel 2000x500 X red; gcBlue=Panel 2000x500 X blue; Color=Black; gcOutColor=Panel 2000x500 X bl
    - DynamicSourceYside_1500 [smart component, from ADD_Library\Recinzione Parametrizzabile.rslib]
        properties: gcBlack=Panel 2000x1500 Y bl; gcYellow=Panel 2000x1500 Y ye; gcRed=Panel 2000x1500 Y red; gcBlue=Panel 2000x1500 Y_blue; Color=Black; gcOutColor=Panel 2000x1500 Y bl
    - DynamicSourceYside_1000 [smart component, from ADD_Library\Recinzione Parametrizzabile.rslib]
        properties: gcBlack=Panel 2000x1000 Y bl; gcYellow=Panel 2000x1000 Y ye; gcRed=Panel 2000x1000 Y red; gcBlue=Panel 2000x1000 Y_blue; Color=Black; gcOutColor=Panel 2000x1000 Y bl
    - DynamicSourceYside_500 [smart component, from ADD_Library\Recinzione Parametrizzabile.rslib]
        properties: gcBlack=Panel 2000x500 Y bl; gcYellow=Panel 2000x500 Y ye; gcRed=Panel 2000x500 Y red; gcBlue=Panel 2000x500 Y blue; Color=Black; gcOutColor=Panel 2000x500 Y bl
    - DynamicSourcePoleXside1 [smart component, from ADD_Library\Recinzione Parametrizzabile.rslib]
        properties: gcBlack=Pole bl; gcYellow=Pole ye; gcRed=Pole_red; gcBlue=Pole_blue; Color=Black; gcOutColor=Pole bl
    - DynamicSourcePoleYside1 [smart component, from ADD_Library\Recinzione Parametrizzabile.rslib]
        properties: gcBlack=PoleYside1 bl; gcYellow=PoleYside1 ye; gcRed=PoleYside1_red; gcBlue=PoleYside1_blue; Color=Black; gcOutColor=PoleYside1 bl
    - DynamicSourcePoleXside2 [smart component, from ADD_Library\Recinzione Parametrizzabile.rslib]
        properties: gcBlack=PoleXside2 bl; gcYellow=PoleXside2 ye; gcRed=PoleXside2_red; gcBlue=PoleXside2_blue; Color=Black; gcOutColor=PoleXside2 bl
    - DynamicSourcePoleYside3 [smart component, from ADD_Library\Recinzione Parametrizzabile.rslib]
        properties: gcBlack=PoleYside3 bl; gcYellow=PoleYside3 ye; gcRed=PoleYside3 red; gcBlue=PoleYside3 blue; Color=Black; gcOutColor=PoleYside3 bl
    - HideObject_1_bl [smart component, from ADD_Library\Recinzione Parametrizzabile.rslib]
        properties: Object=Panel 2000x1500 X bl
    - HideObject_2_bl [smart component, from ADD_Library\Recinzione Parametrizzabile.rslib]
        properties: Object=Panel 2000x1000 X bl
    - HideObject_3_bl [smart component, from ADD_Library\Recinzione Parametrizzabile.rslib]
        properties: Object=Panel 2000x500 X bl
    - HideObject_4_bl [smart component, from ADD_Library\Recinzione Parametrizzabile.rslib]
        properties: Object=Panel 2000x1500 Y bl
    - HideObject_5_bl [smart component, from ADD_Library\Recinzione Parametrizzabile.rslib]
        properties: Object=Panel 2000x1000 Y bl
    - HideObject_6_bl [smart component, from ADD_Library\Recinzione Parametrizzabile.rslib]
        properties: Object=Panel 2000x500 Y bl
    - HideObject_7_bl [smart component, from ADD_Library\Recinzione Parametrizzabile.rslib]
        properties: Object=Pole bl
    - HideObject_8_bl [smart component, from ADD_Library\Recinzione Parametrizzabile.rslib]
        properties: Object=PoleYside1 bl
    - HideObject_9_bl [smart component, from ADD_Library\Recinzione Parametrizzabile.rslib]
        properties: Object=PoleXside2 bl
    - HideObject_10_bl [smart component, from ADD_Library\Recinzione Parametrizzabile.rslib]
        properties: Object=PoleYside3 bl
    - Panel 2000x500 X blue [part, from ADD_Library\Recinzione Parametrizzabile.rslib]
    - Panel 2000x500 X red [part, from ADD_Library\Recinzione Parametrizzabile.rslib]
    - Panel 2000x500 Y blue [part, from ADD_Library\Recinzione Parametrizzabile.rslib]
    - Panel 2000x500 Y red [part, from ADD_Library\Recinzione Parametrizzabile.rslib]
    - Panel 2000x1000 X red [part, from ADD_Library\Recinzione Parametrizzabile.rslib]
    - Panel 2000x1000 X_blue [part, from ADD_Library\Recinzione Parametrizzabile.rslib]
    - Panel 2000x1000 Y red [part, from ADD_Library\Recinzione Parametrizzabile.rslib]
    - Panel 2000x1000 Y_blue [part, from ADD_Library\Recinzione Parametrizzabile.rslib]
    - Panel 2000x1500 X red [part, from ADD_Library\Recinzione Parametrizzabile.rslib]
    - Panel 2000x1500 X_blue [part, from ADD_Library\Recinzione Parametrizzabile.rslib]
    - Panel 2000x1500 Y red [part, from ADD_Library\Recinzione Parametrizzabile.rslib]
    - Panel 2000x1500 Y_blue [part, from ADD_Library\Recinzione Parametrizzabile.rslib]
    - Pole_blue [part, from ADD_Library\Recinzione Parametrizzabile.rslib]
    - Pole_red [part, from ADD_Library\Recinzione Parametrizzabile.rslib]
    - PoleXside2_blue [part, from ADD_Library\Recinzione Parametrizzabile.rslib]
    - PoleXside2_red [part, from ADD_Library\Recinzione Parametrizzabile.rslib]
    - PoleYside1_blue [part, from ADD_Library\Recinzione Parametrizzabile.rslib]
    - PoleYside1_red [part, from ADD_Library\Recinzione Parametrizzabile.rslib]
    - PoleYside3 blue [part, from ADD_Library\Recinzione Parametrizzabile.rslib]
    - PoleYside3 red [part, from ADD_Library\Recinzione Parametrizzabile.rslib]
    - HideObject_red_1 [smart component, from ADD_Library\Recinzione Parametrizzabile.rslib]
        properties: Object=Panel 2000x1500 X red
    - HideObject_red_2 [smart component, from ADD_Library\Recinzione Parametrizzabile.rslib]
        properties: Object=Panel 2000x1500 Y red
    - HideObject_red_3 [smart component, from ADD_Library\Recinzione Parametrizzabile.rslib]
        properties: Object=Panel 2000x1000 X red
    - HideObject_red_4 [smart component, from ADD_Library\Recinzione Parametrizzabile.rslib]
        properties: Object=Panel 2000x1000 Y red
    - HideObject_red_5 [smart component, from ADD_Library\Recinzione Parametrizzabile.rslib]
        properties: Object=Panel 2000x500 X red
    - HideObject_red_6 [smart component, from ADD_Library\Recinzione Parametrizzabile.rslib]
        properties: Object=Panel 2000x500 Y red
    - HideObject_red_7 [smart component, from ADD_Library\Recinzione Parametrizzabile.rslib]
        properties: Object=Pole_red
    - HideObject_red_8 [smart component, from ADD_Library\Recinzione Parametrizzabile.rslib]
        properties: Object=PoleXside2_red
    - HideObject_red_9 [smart component, from ADD_Library\Recinzione Parametrizzabile.rslib]
        properties: Object=PoleYside1_red
    - HideObject_red_10 [smart component, from ADD_Library\Recinzione Parametrizzabile.rslib]
        properties: Object=PoleYside3 red
    - HideObject_blue_1 [smart component, from ADD_Library\Recinzione Parametrizzabile.rslib]
        properties: Object=Panel 2000x1500 X_blue
    - HideObject_blue_2 [smart component, from ADD_Library\Recinzione Parametrizzabile.rslib]
        properties: Object=Panel 2000x1500 Y_blue
    - HideObject_blue_3 [smart component, from ADD_Library\Recinzione Parametrizzabile.rslib]
        properties: Object=Panel 2000x1000 X_blue
    - HideObject_blue_4 [smart component, from ADD_Library\Recinzione Parametrizzabile.rslib]
        properties: Object=Panel 2000x1000 Y_blue
    - HideObject_blue_5 [smart component, from ADD_Library\Recinzione Parametrizzabile.rslib]
        properties: Object=Panel 2000x500 X blue
    - HideObject_blue_6 [smart component, from ADD_Library\Recinzione Parametrizzabile.rslib]
        properties: Object=Panel 2000x500 Y blue
    - HideObject_blue_7 [smart component, from ADD_Library\Recinzione Parametrizzabile.rslib]
        properties: Object=Pole_blue
    - HideObject_blue_8 [smart component, from ADD_Library\Recinzione Parametrizzabile.rslib]
        properties: Object=PoleXside2_blue
    - HideObject_blue_9 [smart component, from ADD_Library\Recinzione Parametrizzabile.rslib]
        properties: Object=PoleYside1_blue
    - HideObject_blue_10 [smart component, from ADD_Library\Recinzione Parametrizzabile.rslib]
        properties: Object=PoleYside3 blue
  - 400_guide [part, from Equipment\Conveyor Guide 400.rslib] at (-2478.87, 1033.07, 0) mm
  - STEEL STAIR [part] at (2707.72, -2498.86, 740) mm, rotated rx 90 ry 0 rz 0 deg

--- Backups/IRB_4600_40kg_2.55m/RAPID/TASK1/PROGMOD/Module1.mod ---
MODULE Module1
    !***********************************************************
    !
    ! Modulo:  Module1
    !
    ! Descrizione:
    !   <Inserire descrizione qui>
    !
    ! Autore: abd99
    !
    ! Versione: 1.0
    !
    !***********************************************************


    !***********************************************************
    !
    ! Procedura main
    !
    !   Questo è il punto di ingresso del programma
    !
    !***********************************************************
    PROC main()
        !Aggiungere il codice in questo punto
    ENDPROC
ENDMODULE
